                    SuppressedNode
                      Call Poner_broca
          Popup Message (haltProgram=false message=Linea17 con chica Terminada! inputType=Text)
          Folder Linea18
            Folder Marcar_puntos
              MoveL speed 100 mm/s, acceleration 500 mm/s^2 (useActiveTCP=true) feature=Base
                Waypoint Linea18_A: TCP in base x=-658.633 y=625.71 z=110.713 mm, rx=-0.2145 ry=-3.1278 rz=-0.004 rad; joints [-48.425, -62.133, 90.617, -28.11, -229.743, 0.749] deg; TCP offset x=0.411 y=-218.298 z=37.994 mm, rx=1.558 ry=-0.1255 rz=0.1212 rad
                Waypoint Linea18_B: TCP in base x=-1149.609 y=625.735 z=110.055 mm, rx=1.1641 ry=-2.9058 rz=0.0105 rad; joints [-36.269, -18.655, 11.335, 7.818, -269.001, 0.894] deg
            Folder AB
              'desbaste_inicial'
              bajada_broca := p[0,0,-0.008,0,0,0]
              barrenos_menos1 := 19
              barreno_actual := 0
              Loop While (checkContinuously=false) expression=barreno_actual≤barrenos_menos1
                Folder Perforacion
                  MoveL speed 100 mm/s, acceleration 500 mm/s^2 (useActiveTCP=true) feature=Base
                    If barreno_actual≟6  or barreno_actual≟13
                      barreno_actual := barreno_actual+1
                    internos := interpolate_pose(Linea18_A, Linea18_B, barreno_actual/barrenos_menos1)
                    Waypoint Waypoint (Variable): variable=internos
                    'desbaste_inicial'
                    bajada_broca := p[0,0,-0.008,0,0,0]
                    bajada := p[0,0,0.008,0,0,0]
                    MoveDirectionNode (selectedDirection=ZMinus toolParams=0.1, 0.15)
                      Until DISTANCE (allowActions=false deceleration=3 distanceNodeType=STOP) Distance=0.071; motionParameters(blendRadius=0)
                    MoveDirectionNode (selectedDirection=ZMinus toolParams=0.001, 0.001)
                      Until TOOL_CONTACT_DETECTION (allowActions=false retraction=0 decelerationAcceleration=0.001 decelerationAngularAcceleration=34.906585)
                    Popup Message (haltProgram=false message=punto contacto alanzdo inputType=Text)
                    MoveDirectionNode (selectedDirection=ZPlus toolParams=0.003, 0.005)
                      Until DISTANCE (allowActions=false deceleration=3 distanceNodeType=STOP) Distance=0.002; motionParameters(blendRadius=0)
                    Wait Sleep waitTime=0.3
                    Set DigitalOutput pin=config_out[1]; digitalValue=1
                    Wait Sleep waitTime=0.3
                    SuppressedNode
                      Loop Counting (count=3) loopVariable=Loop_92
                        bajar := pose_add(get_actual_tcp_pose(), bajada_broca)
                        Waypoint Waypoint (Variable): motionParameters(jointSpeed=1.047198 jointAcceleration=1.396263 cartesianSpeed=0.001 cartesianAcceleration=0.005); variable=bajar
                        subir := pose_sub(get_actual_tcp_pose(), bajada_broca)
                        Waypoint Waypoint (Variable): motionParameters(jointSpeed=1.047198 jointAcceleration=1.396263 cartesianSpeed=0.005 cartesianAcceleration=0.01); variable=subir
                        bajada_broca := pose_sub(bajada_broca, bajada)
                    MoveDirectionNode (selectedDirection=ZPlus toolParams=0.1, 0.15)
                      Until DISTANCE (allowActions=false deceleration=3 distanceNodeType=STOP) Distance=0.08; motionParameters(blendRadius=0)
                    Set DigitalOutput pin=config_out[1]; digitalValue=0
                    barreno_actual := barreno_actual+1
                    SuppressedNode
                      Call Quitar_broca
                    SuppressedNode
                      Call Poner_broca
          Popup Message (haltProgram=false message=Linea18 con chica Terminada! inputType=Text)
      Folder Broca_1
        Folder Linea7
          Folder Marcar_puntos
            MoveL speed 100 mm/s, acceleration 500 mm/s^2 (useActiveTCP=true) feature=Base
              Waypoint Home2: TCP in base x=-476.229 y=0 z=568.737 mm, rx=2.0263 ry=-2.3929 rz=-0.0208 rad; joints [-32.551, -116.469, 98.413, 17.843, -302.102, -0.163] deg; TCP offset x=0.411 y=-218.298 z=37.994 mm, rx=1.558 ry=-0.1255 rz=0.1212 rad
              Waypoint Linea7_A: TCP in base x=-749.561 y=-351.839 z=110.843 mm, rx=3.1084 ry=-0.3759 rz=-0.0174 rad; joints [1.917, -65.95, 96.598, -30.808, -353.455, -0.309] deg
              Folder bajada_comprobacion
                MoveDirectionNode (selectedDirection=ZMinus toolParams=0.1, 0.15)
                  Until DISTANCE (allowActions=false deceleration=3 distanceNodeType=STOP) Distance=0.071; motionParameters(blendRadius=0)
                MoveDirectionNode (selectedDirection=ZMinus toolParams=0.007, 0.007)
                  Until TOOL_CONTACT_DETECTION (allowActions=false retraction=0 decelerationAcceleration=0.02 decelerationAngularAcceleration=34.906585)
                MoveDirectionNode (selectedDirection=ZPlus toolParams=0.1, 0.15)
                  Until DISTANCE (allowActions=false deceleration=3 distanceNodeType=STOP) Distance=0.08; motionParameters(blendRadius=0)
              Waypoint Linea7_B: TCP in base x=-795.37 y=-351.638 z=110.748 mm, rx=3.1084 ry=-0.3758 rz=-0.0174 rad; joints [1.792, -62.243, 90.906, -28.822, -353.578, -0.309] deg
              Folder bajada_comprobacion
                MoveDirectionNode (selectedDirection=ZMinus toolParams=0.1, 0.15)
                  Until DISTANCE (allowActions=false deceleration=3 distanceNodeType=STOP) Distance=0.071; motionParameters(blendRadius=0)
                MoveDirectionNode (selectedDirection=ZMinus toolParams=0.007, 0.007)
                  Until TOOL_CONTACT_DETECTION (allowActions=false retraction=0 decelerationAcceleration=0.02 decelerationAngularAcceleration=34.906585)
                MoveDirectionNode (selectedDirection=ZPlus toolParams=0.1, 0.15)
                  Until DISTANCE (allowActions=false deceleration=3 distanceNodeType=STOP) Distance=0.08; motionParameters(blendRadius=0)
          Folder AB
            'desbaste_inicial'
            bajada_broca := p[0,0,-0.008,0,0,0]
            barrenos_menos1 := 2
            barreno_actual := 0
            Loop While (checkContinuously=false) expression=barreno_actual≤barrenos_menos1
              Folder Perforacion
                MoveL speed 100 mm/s, acceleration 500 mm/s^2 (useActiveTCP=true) feature=Base
                  internos := interpolate_pose(Linea7_A, Linea7_B, barreno_actual/barrenos_menos1)
                  Waypoint Waypoint (Variable): variable=internos
                  'desbaste_inicial'
                  bajada_broca := p[0,0,-0.024,0,0,0]
                  bajada := p[0,0,0.024,0,0,0]
                  MoveDirectionNode (selectedDirection=ZMinus toolParams=0.1, 0.15)
                    Until DISTANCE (allowActions=false deceleration=3 distanceNodeType=STOP) Distance=0.071; motionParameters(blendRadius=0)
                  MoveDirectionNode (selectedDirection=ZMinus toolParams=0.007, 0.007)
                    Until TOOL_CONTACT_DETECTION (allowActions=false retraction=0 decelerationAcceleration=0.02 decelerationAngularAcceleration=34.906585)
                  Popup Message (haltProgram=false message=punto contacto alanzdo inputType=Text)
                  MoveDirectionNode (selectedDirection=ZPlus toolParams=0.003, 0.005)
                    Until DISTANCE (allowActions=false deceleration=3 distanceNodeType=STOP) Distance=0.002; motionParameters(blendRadius=0)
                  Wait Sleep waitTime=0.3
                  Set DigitalOutput pin=config_out[1]; digitalValue=1
                  Wait Sleep waitTime=0.3
                  Loop Counting (count=1) loopVariable(name=Loop_96)
                    bajar := pose_add(get_actual_tcp_pose(), bajada_broca)
                    Waypoint Waypoint (Variable): motionParameters(jointSpeed=1.047198 jointAcceleration=1.396263 cartesianSpeed=0.01 cartesianAcceleration=0.01); variable=bajar
                    subir := pose_sub(get_actual_tcp_pose(), bajada_broca)
                    Waypoint Waypoint (Variable): motionParameters(jointSpeed=1.047198 jointAcceleration=1.396263 cartesianSpeed=0.015 cartesianAcceleration=0.015); variable=subir
                    bajada_broca := pose_sub(bajada_broca, bajada)
                  MoveDirectionNode (selectedDirection=ZPlus toolParams=0.1, 0.15)
                    Until DISTANCE (allowActions=false deceleration=3 distanceNodeType=STOP) Distance=0.08; motionParameters(blendRadius=0)
                  Set DigitalOutput pin=config_out[1]; digitalValue=0
                  barreno_actual := barreno_actual+1
                  Call Quitar_broca
                  Call Poner_broca
        Popup Message (haltProgram=false message=Linea7 con chica Terminada! inputType=Text)
        Folder Linea8
          Folder Marcar_puntos
            MoveL speed 100 mm/s, acceleration 500 mm/s^2 (useActiveTCP=true) feature=Base
              Waypoint Linea8_A: TCP in base x=-897.665 y=-351.421 z=110.406 mm, rx=3.1084 ry=-0.3758 rz=-0.0174 rad; joints [1.574, -53.621, 76.868, -23.4, -353.783, -0.317] deg; TCP offset x=0.411 y=-218.298 z=37.994 mm, rx=1.558 ry=-0.1255 rz=0.1212 rad
              Folder bajada_comprobacion
                MoveDirectionNode (selectedDirection=ZMinus toolParams=0.1, 0.15)
                  Until DISTANCE (allowActions=false deceleration=3 distanceNodeType=STOP) Distance=0.071; motionParameters(blendRadius=0)
                MoveDirectionNode (selectedDirection=ZMinus toolParams=0.007, 0.007)
                  Until TOOL_CONTACT_DETECTION (allowActions=false retraction=0 decelerationAcceleration=0.007 decelerationAngularAcceleration=34.906585)
                MoveDirectionNode (selectedDirection=ZPlus toolParams=0.1, 0.15)
                  Until DISTANCE (allowActions=false deceleration=3 distanceNodeType=STOP) Distance=0.08; motionParameters(blendRadius=0)
              Waypoint Linea8_B: TCP in base x=-1021.743 y=-350.913 z=110.77 mm, rx=3.1084 ry=-0.3758 rz=-0.0173 rad; joints [1.351, -41.656, 55.75, -14.225, -353.984, -0.335] deg; TCP offset x=0.411 y=-218.298 z=37.994 mm, rx=1.558 ry=-0.1255 rz=0.1212 rad
              Folder bajada_comprobacion
                MoveDirectionNode (selectedDirection=ZMinus toolParams=0.1, 0.15)
                  Until DISTANCE (allowActions=false deceleration=3 distanceNodeType=STOP) Distance=0.071; motionParameters(blendRadius=0)
                MoveDirectionNode (selectedDirection=ZMinus toolParams=0.007, 0.007)
                  Until TOOL_CONTACT_DETECTION (allowActions=false retraction=0 decelerationAcceleration=0.007 decelerationAngularAcceleration=34.906585)
                MoveDirectionNode (selectedDirection=ZPlus toolParams=0.1, 0.15)
                  Until DISTANCE (allowActions=false deceleration=3 distanceNodeType=STOP) Distance=0.08; motionParameters(blendRadius=0)
          Folder AB
            'desbaste_inicial'
            bajada_broca := p[0,0,-0.008,0,0,0]
            barrenos_menos1 := 5
            barreno_actual := 0
            Loop While (checkContinuously=false) expression=barreno_actual≤barrenos_menos1
              Folder Perforacion
                MoveL speed 100 mm/s, acceleration 500 mm/s^2 (useActiveTCP=true) feature=Base
                  internos := interpolate_pose(Linea8_A, Linea8_B, barreno_actual/barrenos_menos1)
                  Waypoint Waypoint (Variable): variable=internos
                  'desbaste_inicial'
                  bajada_broca := p[0,0,-0.024,0,0,0]
                  bajada := p[0,0,0.0024,0,0,0]
                  MoveDirectionNode (selectedDirection=ZMinus toolParams=0.1, 0.15)
                    Until DISTANCE (allowActions=false deceleration=3 distanceNodeType=STOP) Distance=0.071; motionParameters(blendRadius=0)
                  MoveDirectionNode (selectedDirection=ZMinus toolParams=0.01, 0.01)
                    Until TOOL_CONTACT_DETECTION (allowActions=false retraction=0 decelerationAcceleration=0.01 decelerationAngularAcceleration=34.906585)
                  Popup Message (haltProgram=false message=punto contacto alanzdo inputType=Text)
                  MoveDirectionNode (selectedDirection=ZPlus toolParams=0.003, 0.005)
                    Until DISTANCE (allowActions=false deceleration=3 distanceNodeType=STOP) Distance=0.002; motionParameters(blendRadius=0)
                  Wait Sleep waitTime=0.3
                  Set DigitalOutput pin=config_out[1]; digitalValue=1
                  Wait Sleep waitTime=0.3
                  Loop Counting (count=1) loopVariable(name=Loop_110)
                    bajar := pose_add(get_actual_tcp_pose(), bajada_broca)
                    Waypoint Waypoint (Variable): motionParameters(jointSpeed=1.047198 jointAcceleration=1.396263 cartesianSpeed=0.01 cartesianAcceleration=0.01); variable=bajar
                    subir := pose_sub(get_actual_tcp_pose(), bajada_broca)
                    Waypoint Waypoint (Variable): motionParameters(jointSpeed=1.047198 jointAcceleration=1.396263 cartesianSpeed=0.015 cartesianAcceleration=0.015); variable=subir
                    bajada_broca := pose_sub(bajada_broca, bajada)
                  MoveDirectionNode (selectedDirection=ZPlus toolParams=0.1, 0.15)
                    Until DISTANCE (allowActions=false deceleration=3 distanceNodeType=STOP) Distance=0.08; motionParameters(blendRadius=0)
                  Set DigitalOutput pin=config_out[1]; digitalValue=0
                  barreno_actual := barreno_actual+1
                  Call Quitar_broca
                  Call Poner_broca
        Popup Message (haltProgram=false message=Linea8 con chica Terminada! inputType=Text)
        Folder Linea9
          Folder Marcar_puntos
            MoveL speed 100 mm/s, acceleration 500 mm/s^2 (useActiveTCP=true) feature=Base
              Waypoint Linea9_A: TCP in base x=-1101.64 y=-350.63 z=110.828 mm, rx=3.1084 ry=-0.3759 rz=-0.0174 rad; joints [1.234, -31.471, 36.669, -5.317, -354.073, -0.351] deg; TCP offset x=0.411 y=-218.298 z=37.994 mm, rx=1.558 ry=-0.1255 rz=0.1212 rad
              Folder bajada_comprobacion
                MoveDirectionNode (selectedDirection=ZMinus toolParams=0.1, 0.15)
                  Until DISTANCE (allowActions=false deceleration=3 distanceNodeType=STOP) Distance=0.071; motionParameters(blendRadius=0)
                MoveDirectionNode (selectedDirection=ZMinus toolParams=0.007, 0.007)
                  Until TOOL_CONTACT_DETECTION (allowActions=false retraction=0 decelerationAcceleration=0.007 decelerationAngularAcceleration=34.906585)
                MoveDirectionNode (selectedDirection=ZPlus toolParams=0.1, 0.15)
                  Until DISTANCE (allowActions=false deceleration=3 distanceNodeType=STOP) Distance=0.08; motionParameters(blendRadius=0)
              Waypoint Linea9_B: TCP in base x=-1151.202 y=-350.816 z=110.405 mm, rx=3.1084 ry=-0.3759 rz=-0.0174 rad; joints [1.184, -21.077, 16.327, 4.623, -354.093, -0.341] deg
              Folder bajada_comprobacion
                MoveDirectionNode (selectedDirection=ZMinus toolParams=0.1, 0.15)
                  Until DISTANCE (allowActions=false deceleration=3 distanceNodeType=STOP) Distance=0.071; motionParameters(blendRadius=0)
                MoveDirectionNode (selectedDirection=ZMinus toolParams=0.007, 0.007)
                  Until TOOL_CONTACT_DETECTION (allowActions=false retraction=0 decelerationAcceleration=0.007 decelerationAngularAcceleration=34.906585)
                MoveDirectionNode (selectedDirection=ZPlus toolParams=0.1, 0.15)
                  Until DISTANCE (allowActions=false deceleration=3 distanceNodeType=STOP) Distance=0.08; motionParameters(blendRadius=0)
          Folder AB
            'desbaste_inicial'
            bajada_broca := p[0,0,-0.008,0,0,0]
            barrenos_menos1 := 2
            barreno_actual := 2
            Loop While (checkContinuously=false) expression=barreno_actual≤barrenos_menos1
              Folder Perforacion
                MoveL speed 100 mm/s, acceleration 500 mm/s^2 (useActiveTCP=true) feature=Base
                  internos := interpolate_pose(Linea9_A, Linea9_B, barreno_actual/barrenos_menos1)
                  Waypoint Waypoint (Variable): variable=internos
                  'desbaste_inicial'
                  bajada_broca := p[0,0,-0.024,0,0,0]
                  bajada := p[0,0,0.024,0,0,0]
                  MoveDirectionNode (selectedDirection=ZMinus toolParams=0.1, 0.15)
                    Until DISTANCE (allowActions=false deceleration=3 distanceNodeType=STOP) Distance=0.071; motionParameters(blendRadius=0)
                  MoveDirectionNode (selectedDirection=ZMinus toolParams=0.01, 0.01)
                    Until TOOL_CONTACT_DETECTION (allowActions=false retraction=0 decelerationAcceleration=0.01 decelerationAngularAcceleration=34.906585)
                  Popup Message (haltProgram=false message=punto contacto alanzdo inputType=Text)
                  MoveDirectionNode (selectedDirection=ZPlus toolParams=0.015, 0.015)
                    Until DISTANCE (allowActions=false deceleration=3 distanceNodeType=STOP) Distance=0.007; motionParameters(blendRadius=0)
                  Wait Sleep waitTime=0.3
                  Set DigitalOutput pin=config_out[1]; digitalValue=1
                  Wait Sleep waitTime=0.3
                  Loop Counting (count=1) loopVariable(name=Loop_114)
                    bajar := pose_add(get_actual_tcp_pose(), bajada_broca)
                    Waypoint Waypoint (Variable): motionParameters(jointSpeed=1.047198 jointAcceleration=1.396263 cartesianSpeed=0.01 cartesianAcceleration=0.01); variable=bajar
                    subir := pose_sub(get_actual_tcp_pose(), bajada_broca)
                    MoveDirectionNode (selectedDirection=ZPlus)
                      Until DISTANCE (allowActions=false deceleration=3 distanceNodeType=STOP) Distance=0.002; motionParameters(blendRadius=0)
                    Set DigitalOutput pin=config_out[1]; digitalValue=0
                    Waypoint Waypoint (Variable): motionParameters(jointSpeed=1.047198 jointAcceleration=1.396263 cartesianSpeed=0.015 cartesianAcceleration=0.015); variable=subir
                    bajada_broca := pose_sub(bajada_broca, bajada)
                  MoveDirectionNode (selectedDirection=ZPlus toolParams=0.1, 0.15)
                    Until DISTANCE (allowActions=false deceleration=3 distanceNodeType=STOP) Distance=0.08; motionParameters(blendRadius=0)
                  Set DigitalOutput pin=config_out[1]; digitalValue=0
                  barreno_actual := barreno_actual+1
                  Call Quitar_broca
                  Call Poner_broca
        Popup Message (haltProgram=false message=Linea9 con chica Terminada! inputType=Text)
        Folder Linea10
          Folder Marcar_puntos
            MoveL speed 100 mm/s, acceleration 500 mm/s^2 (useActiveTCP=true) feature=Base
              Waypoint Home2: TCP in base x=-476.229 y=0 z=568.737 mm, rx=2.0263 ry=-2.3929 rz=-0.0208 rad; joints [-32.551, -116.469, 98.413, 17.843, -302.102, -0.163] deg; TCP offset x=0.411 y=-218.298 z=37.994 mm, rx=1.558 ry=-0.1255 rz=0.1212 rad
              Waypoint Linea10_A: TCP in base x=-633.308 y=-317.691 z=110.995 mm, rx=3.1084 ry=-0.3759 rz=-0.0173 rad; joints [-0.882, -76.128, 110.969, -35.097, -356.258, -0.208] deg
              Folder bajada_comprobacion
                MoveDirectionNode (selectedDirection=ZMinus toolParams=0.1, 0.15)
                  Until DISTANCE (allowActions=false deceleration=3 distanceNodeType=STOP) Distance=0.071; motionParameters(blendRadius=0)
                MoveDirectionNode (selectedDirection=ZMinus toolParams=0.007, 0.007)
                  Until TOOL_CONTACT_DETECTION (allowActions=false retraction=0 decelerationAcceleration=0.02 decelerationAngularAcceleration=34.906585)
                MoveDirectionNode (selectedDirection=ZPlus toolParams=0.1, 0.15)
                  Until DISTANCE (allowActions=false deceleration=3 distanceNodeType=STOP) Distance=0.08; motionParameters(blendRadius=0)
              Waypoint Linea10_B: TCP in base x=-636.724 y=-266.696 z=110.314 mm, rx=2.0205 ry=-2.3939 rz=-0.0206 rad; joints [10.675, -83.921, 120.731, -37.208, -258.826, -0.176] deg
              Folder bajada_comprobacion
                MoveDirectionNode (selectedDirection=ZMinus toolParams=0.1, 0.15)
                  Until DISTANCE (allowActions=false deceleration=3 distanceNodeType=STOP) Distance=0.071; motionParameters(blendRadius=0)
                MoveDirectionNode (selectedDirection=ZMinus toolParams=0.007, 0.007)
                  Until TOOL_CONTACT_DETECTION (allowActions=false retraction=0 decelerationAcceleration=0.02 decelerationAngularAcceleration=34.906585)
                MoveDirectionNode (selectedDirection=ZPlus toolParams=0.1, 0.15)
                  Until DISTANCE (allowActions=false deceleration=3 distanceNodeType=STOP) Distance=0.08; motionParameters(blendRadius=0)
          Folder AB
            'desbaste_inicial'
            bajada_broca := p[0,0,-0.008,0,0,0]
            barrenos_menos1 := 2
            barreno_actual := 0
            Loop While (checkContinuously=false) expression=barreno_actual≤barrenos_menos1
              Folder Perforacion
                MoveL speed 100 mm/s, acceleration 500 mm/s^2 (useActiveTCP=true) feature=Base
                  internos := interpolate_pose(Linea10_A, Linea10_B, barreno_actual/barrenos_menos1)
                  Waypoint Waypoint (Variable): variable=internos
                  'desbaste_inicial'
                  bajada_broca := p[0,0,-0.024,0,0,0]
                  bajada := p[0,0,0.024,0,0,0]
                  MoveDirectionNode (selectedDirection=ZMinus toolParams=0.1, 0.15)
                    Until DISTANCE (allowActions=false deceleration=3 distanceNodeType=STOP) Distance=0.071; motionParameters(blendRadius=0)
                  MoveDirectionNode (selectedDirection=ZMinus toolParams=0.007, 0.007)
                    Until TOOL_CONTACT_DETECTION (allowActions=false retraction=0 decelerationAcceleration=0.02 decelerationAngularAcceleration=34.906585)
                  Popup Message (haltProgram=false message=punto contacto alanzdo inputType=Text)
                  MoveDirectionNode (selectedDirection=ZPlus toolParams=0.015, 0.015)
                    Until DISTANCE (allowActions=false deceleration=3 distanceNodeType=STOP) Distance=0.007; motionParameters(blendRadius=0)
                  Wait Sleep waitTime=0.3
                  Set DigitalOutput pin=config_out[1]; digitalValue=1
                  Wait Sleep waitTime=0.3
                  Loop Counting (count=1) loopVariable(name=Loop_118)
                    bajar := pose_add(get_actual_tcp_pose(), bajada_broca)
                    Waypoint Waypoint (Variable): motionParameters(jointSpeed=1.047198 jointAcceleration=1.396263 cartesianSpeed=0.004 cartesianAcceleration=0.004); variable=bajar
                    subir := pose_sub(get_actual_tcp_pose(), bajada_broca)
                    MoveDirectionNode (selectedDirection=ZPlus toolParams=0.015, 0.015)
                      Until DISTANCE (allowActions=false deceleration=3 distanceNodeType=STOP) Distance=0.002; motionParameters(blendRadius=0)
                    Set DigitalOutput pin=config_out[1]; digitalValue=0
                    Waypoint Waypoint (Variable): motionParameters(jointSpeed=1.047198 jointAcceleration=1.396263 cartesianSpeed=0.015 cartesianAcceleration=0.015); variable=subir
                    bajada_broca := pose_sub(bajada_broca, bajada)
                  MoveDirectionNode (selectedDirection=ZPlus toolParams=0.1, 0.15)
                    Until DISTANCE (allowActions=false deceleration=3 distanceNodeType=STOP) Distance=0.08; motionParameters(blendRadius=0)
                  Set DigitalOutput pin=config_out[1]; digitalValue=0
                  barreno_actual := barreno_actual+1
                  SuppressedNode
                    Call Quitar_broca
                  SuppressedNode
                    Call Poner_broca
        Popup Message (haltProgram=false message=Linea10 con chica Terminada! inputType=Text)
        Folder Linea11
          Folder Marcar_puntos
            MoveL speed 100 mm/s, acceleration 500 mm/s^2 (useActiveTCP=true) feature=Base
              Waypoint Linea11_A: TCP in base x=-635.968 y=-137.768 z=110.292 mm, rx=2.0222 ry=-2.396 rz=-0.017 rad; joints [-4.214, -88.643, 125.799, -37.329, -273.711, -0.094] deg; TCP offset x=0.411 y=-218.298 z=37.994 mm, rx=1.558 ry=-0.1255 rz=0.1212 rad
              Folder bajada_comprobacion
                MoveDirectionNode (selectedDirection=ZMinus toolParams=0.1, 0.15)
                  Until DISTANCE (allowActions=false deceleration=3 distanceNodeType=STOP) Distance=0.071; motionParameters(blendRadius=0)
                MoveDirectionNode (selectedDirection=ZMinus toolParams=0.007, 0.007)
                  Until TOOL_CONTACT_DETECTION (allowActions=false retraction=0 decelerationAcceleration=0.02 decelerationAngularAcceleration=34.906585)
                MoveDirectionNode (selectedDirection=ZPlus toolParams=0.1, 0.15)
                  Until DISTANCE (allowActions=false deceleration=3 distanceNodeType=STOP) Distance=0.08; motionParameters(blendRadius=0)
              Waypoint Linea11_B: TCP in base x=-635.824 y=-83.112 z=110.948 mm, rx=2.0204 ry=-2.3939 rz=-0.0206 rad; joints [-10.934, -90.004, 127.169, -37.541, -280.432, -0.033] deg
              Folder bajada_comprobacion
                MoveDirectionNode (selectedDirection=ZMinus toolParams=0.1, 0.15)
                  Until DISTANCE (allowActions=false deceleration=3 distanceNodeType=STOP) Distance=0.071; motionParameters(blendRadius=0)
                MoveDirectionNode (selectedDirection=ZMinus toolParams=0.007, 0.007)
                  Until TOOL_CONTACT_DETECTION (allowActions=false retraction=0 decelerationAcceleration=0.02 decelerationAngularAcceleration=34.906585)
                MoveDirectionNode (selectedDirection=ZPlus toolParams=0.1, 0.15)
                  Until DISTANCE (allowActions=false deceleration=3 distanceNodeType=STOP) Distance=0.08; motionParameters(blendRadius=0)
          Folder AB
            'desbaste_inicial'
            bajada_broca := p[0,0,-0.008,0,0,0]
            barrenos_menos1 := 2
            barreno_actual := 0
            Loop While (checkContinuously=false) expression=barreno_actual≤barrenos_menos1
              Folder Perforacion
                MoveL speed 100 mm/s, acceleration 500 mm/s^2 (useActiveTCP=true) feature=Base
                  SuppressedNode
                    If barreno_actual≟5
                      barreno_actual := barreno_actual+1
                  internos := interpolate_pose(Linea11_A, Linea11_B, barreno_actual/barrenos_menos1)
                  Waypoint Waypoint (Variable): variable=internos
                  'desbaste_inicial'
                  bajada_broca := p[0,0,-0.024,0,0,0]
                  bajada := p[0,0,0.024,0,0,0]
                  MoveDirectionNode (selectedDirection=ZMinus toolParams=0.1, 0.15)
                    Until DISTANCE (allowActions=false deceleration=3 distanceNodeType=STOP) Distance=0.071; motionParameters(blendRadius=0)
                  MoveDirectionNode (selectedDirection=ZMinus toolParams=0.007, 0.007)
                    Until TOOL_CONTACT_DETECTION (allowActions=false retraction=0 decelerationAcceleration=0.02 decelerationAngularAcceleration=34.906585)
                  Popup Message (haltProgram=false message=punto contacto alanzdo inputType=Text)
                  MoveDirectionNode (selectedDirection=ZPlus toolParams=0.015, 0.015)
                    Until DISTANCE (allowActions=false deceleration=3 distanceNodeType=STOP) Distance=0.007; motionParameters(blendRadius=0)
                  Wait Sleep waitTime=0.3
                  Set DigitalOutput pin=config_out[1]; digitalValue=1
                  Wait Sleep waitTime=0.3
                  Loop Counting (count=1) loopVariable(name=Loop_122)
                    bajar := pose_add(get_actual_tcp_pose(), bajada_broca)
                    Waypoint Waypoint (Variable): motionParameters(jointSpeed=1.047198 jointAcceleration=1.396263 cartesianSpeed=0.004 cartesianAcceleration=0.004); variable=bajar
                    subir := pose_sub(get_actual_tcp_pose(), bajada_broca)
                    MoveDirectionNode (selectedDirection=ZPlus toolParams=0.015, 0.015)
                      Until DISTANCE (allowActions=false deceleration=3 distanceNodeType=STOP) Distance=0.002; motionParameters(blendRadius=0)
                    Set DigitalOutput pin=config_out[1]; digitalValue=0
                    Waypoint Waypoint (Variable): motionParameters(jointSpeed=1.047198 jointAcceleration=1.396263 cartesianSpeed=0.015 cartesianAcceleration=0.015); variable=subir
                    bajada_broca := pose_sub(bajada_broca, bajada)
                  MoveDirectionNode (selectedDirection=ZPlus toolParams=0.1, 0.15)
                    Until DISTANCE (allowActions=false deceleration=3 distanceNodeType=STOP) Distance=0.08; motionParameters(blendRadius=0)
                  Set DigitalOutput pin=config_out[1]; digitalValue=0
                  barreno_actual := barreno_actual+1
                  SuppressedNode
                    Call Quitar_broca
                  SuppressedNode
                    Call Poner_broca
        Popup Message (haltProgram=false message=Linea11 con chica Terminada! inputType=Text)
        Folder Linea12
          Folder Marcar_puntos
            MoveL speed 100 mm/s, acceleration 500 mm/s^2 (useActiveTCP=true) feature=Base
              Waypoint Linea12_A: TCP in base x=-635.349 y=-59.56 z=110.675 mm, rx=2.0204 ry=-2.3939 rz=-0.0205 rad; joints [-13.849, -90.386, 127.583, -37.571, -283.348, -0.016] deg
              Folder bajada_comprobacion
                MoveDirectionNode (selectedDirection=ZMinus toolParams=0.1, 0.15)
                  Until DISTANCE (allowActions=false deceleration=3 distanceNodeType=STOP) Distance=0.071; motionParameters(blendRadius=0)
                MoveDirectionNode (selectedDirection=ZMinus toolParams=0.007, 0.007)
                  Until TOOL_CONTACT_DETECTION (allowActions=false retraction=0 decelerationAcceleration=0.02 decelerationAngularAcceleration=34.906585)
                MoveDirectionNode (selectedDirection=ZPlus toolParams=0.1, 0.15)
                  Until DISTANCE (allowActions=false deceleration=3 distanceNodeType=STOP) Distance=0.08; motionParameters(blendRadius=0)
              Waypoint Linea12_B: TCP in base x=-634.713 y=114.181 z=110.553 mm, rx=2.0204 ry=-2.3939 rz=-0.0206 rad; joints [-33.919, -89.532, 126.745, -37.627, -303.419, 0.135] deg
              Folder bajada_comprobacion
                MoveDirectionNode (selectedDirection=ZMinus toolParams=0.1, 0.15)
                  Until DISTANCE (allowActions=false deceleration=3 distanceNodeType=STOP) Distance=0.071; motionParameters(blendRadius=0)
                MoveDirectionNode (selectedDirection=ZMinus toolParams=0.007, 0.007)
                  Until TOOL_CONTACT_DETECTION (allowActions=false retraction=0 decelerationAcceleration=0.02 decelerationAngularAcceleration=34.906585)
                MoveDirectionNode (selectedDirection=ZPlus toolParams=0.1, 0.15)
                  Until DISTANCE (allowActions=false deceleration=3 distanceNodeType=STOP) Distance=0.08; motionParameters(blendRadius=0)
          Folder AB
            'desbaste_inicial'
            bajada_broca := p[0,0,-0.008,0,0,0]
            barrenos_menos1 := 7
            barreno_actual := 0
            Loop While (checkContinuously=false) expression=barreno_actual≤barrenos_menos1
              Folder Perforacion
                MoveL speed 100 mm/s, acceleration 500 mm/s^2 (useActiveTCP=true) feature=Base
                  If barreno_actual≟2
                    barreno_actual := barreno_actual+1
                  internos := interpolate_pose(Linea12_A, Linea12_B, barreno_actual/barrenos_menos1)
                  Waypoint Waypoint (Variable): variable=internos
                  'desbaste_inicial'
                  bajada_broca := p[0,0,-0.024,0,0,0]
                  bajada := p[0,0,0.024,0,0,0]
                  MoveDirectionNode (selectedDirection=ZMinus toolParams=0.1, 0.15)
                    Until DISTANCE (allowActions=false deceleration=3 distanceNodeType=STOP) Distance=0.071; motionParameters(blendRadius=0)
                  MoveDirectionNode (selectedDirection=ZMinus toolParams=0.007, 0.007)
                    Until TOOL_CONTACT_DETECTION (allowActions=false retraction=0 decelerationAcceleration=0.02 decelerationAngularAcceleration=34.906585)
                  Popup Message (haltProgram=false message=punto contacto alanzdo inputType=Text)
                  MoveDirectionNode (selectedDirection=ZPlus toolParams=0.003, 0.005)
                    Until DISTANCE (allowActions=false deceleration=3 distanceNodeType=STOP) Distance=0.002; motionParameters(blendRadius=0)
                  Wait Sleep waitTime=0.3
                  Set DigitalOutput pin=config_out[1]; digitalValue=1
                  Wait Sleep waitTime=0.3
                  Loop Counting (count=1) loopVariable(name=Loop_126)
                    bajar := pose_add(get_actual_tcp_pose(), bajada_broca)
                    Waypoint Waypoint (Variable): motionParameters(jointSpeed=1.047198 jointAcceleration=1.396263 cartesianSpeed=0.004 cartesianAcceleration=0.004); variable=bajar
                    subir := pose_sub(get_actual_tcp_pose(), bajada_broca)
                    MoveDirectionNode (selectedDirection=ZPlus toolParams=0.015, 0.015)
                      Until DISTANCE (allowActions=false deceleration=3 distanceNodeType=STOP) Distance=0.002; motionParameters(blendRadius=0)
                    Set DigitalOutput pin=config_out[1]; digitalValue=0
                    Waypoint Waypoint (Variable): motionParameters(jointSpeed=1.047198 jointAcceleration=1.396263 cartesianSpeed=0.015 cartesianAcceleration=0.015); variable=subir
                    bajada_broca := pose_sub(bajada_broca, bajada)
                  MoveDirectionNode (selectedDirection=ZPlus toolParams=0.1, 0.15)
                    Until DISTANCE (allowActions=false deceleration=3 distanceNodeType=STOP) Distance=0.08; motionParameters(blendRadius=0)
                  Set DigitalOutput pin=config_out[1]; digitalValue=0
                  barreno_actual := barreno_actual+1
                  SuppressedNode
                    Call Quitar_broca
                  SuppressedNode
                    Call Poner_broca
        Popup Message (haltProgram=false message=Linea12 con chica Terminada! inputType=Text)
        Folder Linea13
          Folder Marcar_puntos
            MoveL speed 100 mm/s, acceleration 500 mm/s^2 (useActiveTCP=true) feature=Base
              Waypoint Linea13_A: TCP in base x=-634.623 y=269.838 z=110.202 mm, rx=2.0205 ry=-2.3939 rz=-0.0206 rad; joints [-47.693, -84.101, 120.951, -37.343, -317.193, 0.28] deg
              Folder bajada_comprobacion
                MoveDirectionNode (selectedDirection=ZMinus toolParams=0.1, 0.15)
                  Until DISTANCE (allowActions=false deceleration=3 distanceNodeType=STOP) Distance=0.071; motionParameters(blendRadius=0)
                MoveDirectionNode (selectedDirection=ZMinus toolParams=0.007, 0.007)
                  Until TOOL_CONTACT_DETECTION (allowActions=false retraction=0 decelerationAcceleration=0.02 decelerationAngularAcceleration=34.906585)
                MoveDirectionNode (selectedDirection=ZPlus toolParams=0.1, 0.15)
                  Until DISTANCE (allowActions=false deceleration=3 distanceNodeType=STOP) Distance=0.08; motionParameters(blendRadius=0)
              Waypoint Linea13_B: TCP in base x=-634.043 y=326.314 z=110.496 mm, rx=2.0205 ry=-2.3939 rz=-0.0206 rad; joints [-51.641, -81.48, 117.853, -36.903, -321.141, 0.338] deg
              Folder bajada_comprobacion
                MoveDirectionNode (selectedDirection=ZMinus toolParams=0.1, 0.15)
                  Until DISTANCE (allowActions=false deceleration=3 distanceNodeType=STOP) Distance=0.071; motionParameters(blendRadius=0)
                MoveDirectionNode (selectedDirection=ZMinus toolParams=0.007, 0.007)
                  Until TOOL_CONTACT_DETECTION (allowActions=false retraction=0 decelerationAcceleration=0.02 decelerationAngularAcceleration=34.906585)
                MoveDirectionNode (selectedDirection=ZPlus toolParams=0.1, 0.15)
                  Until DISTANCE (allowActions=false deceleration=3 distanceNodeType=STOP) Distance=0.08; motionParameters(blendRadius=0)
          Folder AB
            'desbaste_inicial'
            bajada_broca := p[0,0,-0.008,0,0,0]
            barrenos_menos1 := 2
            barreno_actual := 0
            Loop While (checkContinuously=false) expression=barreno_actual≤barrenos_menos1
              Folder Perforacion
                MoveL speed 100 mm/s, acceleration 500 mm/s^2 (useActiveTCP=true) feature=Base
                  SuppressedNode
                    If barreno_actual≟2
                      barreno_actual := barreno_actual+1
                  internos := interpolate_pose(Linea13_A, Linea13_B, barreno_actual/barrenos_menos1)
                  Waypoint Waypoint (Variable): variable=internos
                  'desbaste_inicial'
                  bajada_broca := p[0,0,-0.024,0,0,0]
                  bajada := p[0,0,0.024,0,0,0]
                  MoveDirectionNode (selectedDirection=ZMinus toolParams=0.1, 0.15)
                    Until DISTANCE (allowActions=false deceleration=3 distanceNodeType=STOP) Distance=0.071; motionParameters(blendRadius=0)
                  MoveDirectionNode (selectedDirection=ZMinus toolParams=0.007, 0.007)
                    Until TOOL_CONTACT_DETECTION (allowActions=false retraction=0 decelerationAcceleration=0.02 decelerationAngularAcceleration=34.906585)
                  Popup Message (haltProgram=false message=punto contacto alanzdo inputType=Text)
                  MoveDirectionNode (selectedDirection=ZPlus toolParams=0.003, 0.005)
                    Until DISTANCE (allowActions=false deceleration=3 distanceNodeType=STOP) Distance=0.002; motionParameters(blendRadius=0)
                  Wait Sleep waitTime=0.3
                  Set DigitalOutput pin=config_out[1]; digitalValue=1
                  Wait Sleep waitTime=0.3
                  Loop Counting (count=1) loopVariable(name=Loop_129)
                    bajar := pose_add(get_actual_tcp_pose(), bajada_broca)
                    Waypoint Waypoint (Variable): motionParameters(jointSpeed=1.047198 jointAcceleration=1.396263 cartesianSpeed=0.004 cartesianAcceleration=0.004); variable=bajar
                    subir := pose_sub(get_actual_tcp_pose(), bajada_broca)
                    MoveDirectionNode (selectedDirection=ZPlus toolParams=0.015, 0.015)
                      Until DISTANCE (allowActions=false deceleration=3 distanceNodeType=STOP) Distance=0.002; motionParameters(blendRadius=0)
                    Set DigitalOutput pin=config_out[1]; digitalValue=0
                    Waypoint Waypoint (Variable): motionParameters(jointSpeed=1.047198 jointAcceleration=1.396263 cartesianSpeed=0.015 cartesianAcceleration=0.015); variable=subir
                    bajada_broca := pose_sub(bajada_broca, bajada)
                  MoveDirectionNode (selectedDirection=ZPlus toolParams=0.1, 0.15)
                    Until DISTANCE (allowActions=false deceleration=3 distanceNodeType=STOP) Distance=0.08; motionParameters(blendRadius=0)
                  Set DigitalOutput pin=config_out[1]; digitalValue=0
                  barreno_actual := barreno_actual+1
                  SuppressedNode
                    Call Quitar_broca
                  SuppressedNode
                    Call Poner_broca
        Popup Message (haltProgram=false message=Linea13 con chica Terminada! inputType=Text)
        Folder Linea14
          Folder Marcar_puntos
            MoveL speed 100 mm/s, acceleration 500 mm/s^2 (useActiveTCP=true) feature=Base
              Waypoint Linea14_A: TCP in base x=-633.963 y=349.887 z=111.384 mm, rx=2.0205 ry=-2.3938 rz=-0.0205 rad; joints [-53.122, -80.339, 116.362, -36.569, -322.623, 0.363] deg
              Folder bajada_comprobacion
                MoveDirectionNode (selectedDirection=ZMinus toolParams=0.1, 0.15)
                  Until DISTANCE (allowActions=false deceleration=3 distanceNodeType=STOP) Distance=0.071; motionParameters(blendRadius=0)
                MoveDirectionNode (selectedDirection=ZMinus toolParams=0.007, 0.007)
                  Until TOOL_CONTACT_DETECTION (allowActions=false retraction=0 decelerationAcceleration=0.02 decelerationAngularAcceleration=34.906585)
                MoveDirectionNode (selectedDirection=ZPlus toolParams=0.1, 0.15)
                  Until DISTANCE (allowActions=false deceleration=3 distanceNodeType=STOP) Distance=0.08; motionParameters(blendRadius=0)
              Waypoint Linea14_B: TCP in base x=-633.711 y=491.848 z=110.684 mm, rx=2.0205 ry=-2.3939 rz=-0.0205 rad; joints [-60.395, -72.347, 105.992, -34.301, -329.892, 0.503] deg
              Folder bajada_comprobacion
                MoveDirectionNode (selectedDirection=ZMinus toolParams=0.1, 0.15)
                  Until DISTANCE (allowActions=false deceleration=3 distanceNodeType=STOP) Distance=0.071; motionParameters(blendRadius=0)
                MoveDirectionNode (selectedDirection=ZMinus toolParams=0.007, 0.007)
                  Until TOOL_CONTACT_DETECTION (allowActions=false retraction=0 decelerationAcceleration=0.02 decelerationAngularAcceleration=34.906585)
                MoveDirectionNode (selectedDirection=ZPlus toolParams=0.1, 0.15)
                  Until DISTANCE (allowActions=false deceleration=3 distanceNodeType=STOP) Distance=0.08; motionParameters(blendRadius=0)
          Folder AB
            'desbaste_inicial'
            bajada_broca := p[0,0,-0.008,0,0,0]
            barrenos_menos1 := 5
            barreno_actual := 0
            Loop While (checkContinuously=false) expression=barreno_actual≤barrenos_menos1
              Folder Perforacion
                MoveL speed 100 mm/s, acceleration 500 mm/s^2 (useActiveTCP=true) feature=Base
                  If barreno_actual≟3
                    barreno_actual := barreno_actual+1
                  internos := interpolate_pose(Linea14_A, Linea14_B, barreno_actual/barrenos_menos1)
                  Waypoint Waypoint (Variable): variable=internos
                  'desbaste_inicial'
                  bajada_broca := p[0,0,-0.024,0,0,0]
                  bajada := p[0,0,0.024,0,0,0]
                  MoveDirectionNode (selectedDirection=ZMinus toolParams=0.1, 0.15)
                    Until DISTANCE (allowActions=false deceleration=3 distanceNodeType=STOP) Distance=0.071; motionParameters(blendRadius=0)
                  MoveDirectionNode (selectedDirection=ZMinus toolParams=0.007, 0.007)
                    Until TOOL_CONTACT_DETECTION (allowActions=false retraction=0 decelerationAcceleration=0.02 decelerationAngularAcceleration=34.906585)
                  Popup Message (haltProgram=false message=punto contacto alanzdo inputType=Text)
                  MoveDirectionNode (selectedDirection=ZPlus toolParams=0.003, 0.005)
                    Until DISTANCE (allowActions=false deceleration=3 distanceNodeType=STOP) Distance=0.002; motionParameters(blendRadius=0)
                  Wait Sleep waitTime=0.3
                  Set DigitalOutput pin=config_out[1]; digitalValue=1
                  Wait Sleep waitTime=0.3
                  Loop Counting (count=1) loopVariable(name=Loop_131)
                    bajar := pose_add(get_actual_tcp_pose(), bajada_broca)
                    Waypoint Waypoint (Variable): motionParameters(jointSpeed=1.047198 jointAcceleration=1.396263 cartesianSpeed=0.004 cartesianAcceleration=0.004); variable=bajar
                    subir := pose_sub(get_actual_tcp_pose(), bajada_broca)
                    MoveDirectionNode (selectedDirection=ZPlus toolParams=0.015, 0.015)
                      Until DISTANCE (allowActions=false deceleration=3 distanceNodeType=STOP) Distance=0.002; motionParameters(blendRadius=0)
                    Set DigitalOutput pin=config_out[1]; digitalValue=0
                    Waypoint Waypoint (Variable): motionParameters(jointSpeed=1.047198 jointAcceleration=1.396263 cartesianSpeed=0.015 cartesianAcceleration=0.015); variable=subir
                    bajada_broca := pose_sub(bajada_broca, bajada)
                  MoveDirectionNode (selectedDirection=ZPlus toolParams=0.1, 0.15)
                    Until DISTANCE (allowActions=false deceleration=3 distanceNodeType=STOP) Distance=0.08; motionParameters(blendRadius=0)
                  Set DigitalOutput pin=config_out[1]; digitalValue=0
                  barreno_actual := barreno_actual+1
                  SuppressedNode
                    Call Quitar_broca
                  SuppressedNode
                    Call Poner_broca
        Popup Message (haltProgram=false message=Linea14 con chica Terminada! inputType=Text)
        Folder Linea15
          Folder Marcar_puntos
            MoveL speed 100 mm/s, acceleration 500 mm/s^2 (useActiveTCP=true) feature=Base
              Waypoint Linea15_A: TCP in base x=-633.318 y=515.44 z=110.158 mm, rx=2.0204 ry=-2.394 rz=-0.0205 rad; joints [-61.401, -70.918, 104.049, -33.805, -330.892, 0.526] deg
              Folder bajada_comprobacion
                MoveDirectionNode (selectedDirection=ZMinus toolParams=0.1, 0.15)
                  Until DISTANCE (allowActions=false deceleration=3 distanceNodeType=STOP) Distance=0.071; motionParameters(blendRadius=0)
                MoveDirectionNode (selectedDirection=ZMinus toolParams=0.007, 0.007)
                  Until TOOL_CONTACT_DETECTION (allowActions=false retraction=0 decelerationAcceleration=0.02 decelerationAngularAcceleration=34.906585)
                MoveDirectionNode (selectedDirection=ZPlus toolParams=0.1, 0.15)
                  Until DISTANCE (allowActions=false deceleration=3 distanceNodeType=STOP) Distance=0.08; motionParameters(blendRadius=0)
              Waypoint Linea15_B: TCP in base x=-632.971 y=593.971 z=110.611 mm, rx=2.0204 ry=-2.3939 rz=-0.0206 rad; joints [-64.313, -66.034, 96.849, -31.559, -333.804, 0.606] deg
              Folder bajada_comprobacion
                MoveDirectionNode (selectedDirection=ZMinus toolParams=0.1, 0.15)
                  Until DISTANCE (allowActions=false deceleration=3 distanceNodeType=STOP) Distance=0.071; motionParameters(blendRadius=0)
                MoveDirectionNode (selectedDirection=ZMinus toolParams=0.007, 0.007)
                  Until TOOL_CONTACT_DETECTION (allowActions=false retraction=0 decelerationAcceleration=0.02 decelerationAngularAcceleration=34.906585)
                MoveDirectionNode (selectedDirection=ZPlus toolParams=0.1, 0.15)
                  Until DISTANCE (allowActions=false deceleration=3 distanceNodeType=STOP) Distance=0.08; motionParameters(blendRadius=0)
          Folder AB
            'desbaste_inicial'
            bajada_broca := p[0,0,-0.008,0,0,0]
            barrenos_menos1 := 3
            barreno_actual := 0
            Loop While (checkContinuously=false) expression=barreno_actual≤barrenos_menos1
              Folder Perforacion
                MoveL speed 100 mm/s, acceleration 500 mm/s^2 (useActiveTCP=true) feature=Base
                  SuppressedNode
                    If barreno_actual≟3
                      barreno_actual := barreno_actual+1
                  internos := interpolate_pose(Linea15_A, Linea15_B, barreno_actual/barrenos_menos1)
                  Waypoint Waypoint (Variable): variable=internos
                  'desbaste_inicial'
                  bajada_broca := p[0,0,-0.024,0,0,0]
                  bajada := p[0,0,0.024,0,0,0]
                  MoveDirectionNode (selectedDirection=ZMinus toolParams=0.1, 0.15)
                    Until DISTANCE (allowActions=false deceleration=3 distanceNodeType=STOP) Distance=0.071; motionParameters(blendRadius=0)
                  MoveDirectionNode (selectedDirection=ZMinus toolParams=0.007, 0.007)
                    Until TOOL_CONTACT_DETECTION (allowActions=false retraction=0 decelerationAcceleration=0.02 decelerationAngularAcceleration=34.906585)
                  Popup Message (haltProgram=false message=punto contacto alanzdo inputType=Text)
                  MoveDirectionNode (selectedDirection=ZPlus toolParams=0.003, 0.005)
                    Until DISTANCE (allowActions=false deceleration=3 distanceNodeType=STOP) Distance=0.002; motionParameters(blendRadius=0)
                  Wait Sleep waitTime=0.3
                  Set DigitalOutput pin=config_out[1]; digitalValue=1
                  Wait Sleep waitTime=0.3
                  Loop Counting (count=1) loopVariable(name=Loop_133)
                    bajar := pose_add(get_actual_tcp_pose(), bajada_broca)
                    Waypoint Waypoint (Variable): motionParameters(jointSpeed=1.047198 jointAcceleration=1.396263 cartesianSpeed=0.004 cartesianAcceleration=0.004); variable=bajar
                    subir := pose_sub(get_actual_tcp_pose(), bajada_broca)
                    MoveDirectionNode (selectedDirection=ZPlus toolParams=0.015, 0.015)
                      Until DISTANCE (allowActions=false deceleration=3 distanceNodeType=STOP) Distance=0.002; motionParameters(blendRadius=0)
                    Set DigitalOutput pin=config_out[1]; digitalValue=0
                    Waypoint Waypoint (Variable): motionParameters(jointSpeed=1.047198 jointAcceleration=1.396263 cartesianSpeed=0.015 cartesianAcceleration=0.015); variable=subir
                    bajada_broca := pose_sub(bajada_broca, bajada)
                  MoveDirectionNode (selectedDirection=ZPlus toolParams=0.1, 0.15)
                    Until DISTANCE (allowActions=false deceleration=3 distanceNodeType=STOP) Distance=0.08; motionParameters(blendRadius=0)
                  Set DigitalOutput pin=config_out[1]; digitalValue=0
                  barreno_actual := barreno_actual+1
                  SuppressedNode
                    Call Quitar_broca
                  SuppressedNode
                    Call Poner_broca
        Popup Message (haltProgram=false message=Linea15 con chica Terminada! inputType=Text)
        Folder Linea16
          Folder Marcar_puntos
            MoveL speed 100 mm/s, acceleration 500 mm/s^2 (useActiveTCP=true) feature=Base
              Waypoint Linea16_A: TCP in base x=-469.659 y=618.24 z=110.223 mm, rx=-0.2145 ry=-3.1278 rz=-0.004 rad; joints [-60.494, -74.578, 108.875, -33.964, -241.822, 0.658] deg
              Folder bajada_comprobacion
                MoveDirectionNode (selectedDirection=ZMinus toolParams=0.1, 0.15)
                  Until DISTANCE (allowActions=false deceleration=3 distanceNodeType=STOP) Distance=0.071; motionParameters(blendRadius=0)
                MoveDirectionNode (selectedDirection=ZMinus toolParams=0.007, 0.007)
                  Until TOOL_CONTACT_DETECTION (allowActions=false retraction=0 decelerationAcceleration=0.02 decelerationAngularAcceleration=34.906585)
                MoveDirectionNode (selectedDirection=ZPlus toolParams=0.1, 0.15)
                  Until DISTANCE (allowActions=false deceleration=3 distanceNodeType=STOP) Distance=0.08; motionParameters(blendRadius=0)
              Waypoint Linea16_B: TCP in base x=-493.719 y=618.586 z=110.183 mm, rx=-0.2145 ry=-3.1278 rz=-0.004 rad; joints [-58.661, -73.102, 106.872, -33.43, -239.985, 0.672] deg
              Folder bajada_comprobacion
                MoveDirectionNode (selectedDirection=ZMinus toolParams=0.1, 0.15)
                  Until DISTANCE (allowActions=false deceleration=3 distanceNodeType=STOP) Distance=0.071; motionParameters(blendRadius=0)
                MoveDirectionNode (selectedDirection=ZMinus toolParams=0.007, 0.007)
                  Until TOOL_CONTACT_DETECTION (allowActions=false retraction=0 decelerationAcceleration=0.02 decelerationAngularAcceleration=34.906585)
                MoveDirectionNode (selectedDirection=ZPlus toolParams=0.1, 0.15)
                  Until DISTANCE (allowActions=false deceleration=3 distanceNodeType=STOP) Distance=0.08; motionParameters(blendRadius=0)
          Folder AB
            'desbaste_inicial'
            bajada_broca := p[0,0,-0.008,0,0,0]
            barrenos_menos1 := 1
            barreno_actual := 0
            Loop While (checkContinuously=false) expression=barreno_actual≤barrenos_menos1
              Folder Perforacion
                MoveL speed 100 mm/s, acceleration 500 mm/s^2 (useActiveTCP=true) feature=Base
                  SuppressedNode
                    If barreno_actual≟3
                      barreno_actual := barreno_actual+1
                  internos := interpolate_pose(Linea16_A, Linea16_B, barreno_actual/barrenos_menos1)
                  Waypoint Waypoint (Variable): variable=internos
                  'desbaste_inicial'
                  bajada_broca := p[0,0,-0.024,0,0,0]
                  bajada := p[0,0,0.024,0,0,0]
                  MoveDirectionNode (selectedDirection=ZMinus toolParams=0.1, 0.15)
                    Until DISTANCE (allowActions=false deceleration=3 distanceNodeType=STOP) Distance=0.071; motionParameters(blendRadius=0)
                  MoveDirectionNode (selectedDirection=ZMinus toolParams=0.007, 0.007)
                    Until TOOL_CONTACT_DETECTION (allowActions=false retraction=0 decelerationAcceleration=0.02 decelerationAngularAcceleration=34.906585)
                  Popup Message (haltProgram=false message=punto contacto alanzdo inputType=Text)
                  MoveDirectionNode (selectedDirection=ZPlus toolParams=0.003, 0.005)
                    Until DISTANCE (allowActions=false deceleration=3 distanceNodeType=STOP) Distance=0.002; motionParameters(blendRadius=0)
                  Wait Sleep waitTime=0.3
                  Set DigitalOutput pin=config_out[1]; digitalValue=1
                  Wait Sleep waitTime=0.3
                  Loop Counting (count=1) loopVariable(name=Loop_135)
                    bajar := pose_add(get_actual_tcp_pose(), bajada_broca)
                    Waypoint Waypoint (Variable): motionParameters(jointSpeed=1.047198 jointAcceleration=1.396263 cartesianSpeed=0.004 cartesianAcceleration=0.004); variable=bajar
                    subir := pose_sub(get_actual_tcp_pose(), bajada_broca)
                    MoveDirectionNode (selectedDirection=ZPlus toolParams=0.015, 0.015)
                      Until DISTANCE (allowActions=false deceleration=3 distanceNodeType=STOP) Distance=0.002; motionParameters(blendRadius=0)
                    Set DigitalOutput pin=config_out[1]; digitalValue=0
                    Waypoint Waypoint (Variable): motionParameters(jointSpeed=1.047198 jointAcceleration=1.396263 cartesianSpeed=0.015 cartesianAcceleration=0.015); variable=subir
                    bajada_broca := pose_sub(bajada_broca, bajada)
                  MoveDirectionNode (selectedDirection=ZPlus toolParams=0.1, 0.15)
                    Until DISTANCE (allowActions=false deceleration=3 distanceNodeType=STOP) Distance=0.08; motionParameters(blendRadius=0)
                  Set DigitalOutput pin=config_out[1]; digitalValue=0
                  barreno_actual := barreno_actual+1
                  SuppressedNode
                    Call Quitar_broca
                  SuppressedNode
                    Call Poner_broca
        Popup Message (haltProgram=false message=Linea16 con chica Terminada! inputType=Text)
        Folder Linea17
          Folder Marcar_puntos
            MoveL speed 100 mm/s, acceleration 500 mm/s^2 (useActiveTCP=true) feature=Base
              Waypoint Linea17_A: TCP in base x=-523.229 y=618.283 z=110.575 mm, rx=-0.2145 ry=-3.1278 rz=-0.0039 rad; joints [-56.495, -71.324, 104.348, -32.678, -237.82, 0.686] deg
              Folder bajada_comprobacion
                MoveDirectionNode (selectedDirection=ZMinus toolParams=0.1, 0.15)
                  Until DISTANCE (allowActions=false deceleration=3 distanceNodeType=STOP) Distance=0.071; motionParameters(blendRadius=0)
                MoveDirectionNode (selectedDirection=ZMinus toolParams=0.007, 0.007)
                  Until TOOL_CONTACT_DETECTION (allowActions=false retraction=0 decelerationAcceleration=0.02 decelerationAngularAcceleration=34.906585)
                MoveDirectionNode (selectedDirection=ZPlus toolParams=0.1, 0.15)
                  Until DISTANCE (allowActions=false deceleration=3 distanceNodeType=STOP) Distance=0.08; motionParameters(blendRadius=0)
              Waypoint Linea17_B: TCP in base x=-574.505 y=618.78 z=110.128 mm, rx=-0.2145 ry=-3.1278 rz=-0.0039 rad; joints [-53.062, -68.029, 99.656, -31.269, -234.384, 0.712] deg
              Folder bajada_comprobacion
                MoveDirectionNode (selectedDirection=ZMinus toolParams=0.1, 0.15)
                  Until DISTANCE (allowActions=false deceleration=3 distanceNodeType=STOP) Distance=0.071; motionParameters(blendRadius=0)
                MoveDirectionNode (selectedDirection=ZMinus toolParams=0.007, 0.007)
                  Until TOOL_CONTACT_DETECTION (allowActions=false retraction=0 decelerationAcceleration=0.02 decelerationAngularAcceleration=34.906585)
                MoveDirectionNode (selectedDirection=ZPlus toolParams=0.1, 0.15)
                  Until DISTANCE (allowActions=false deceleration=3 distanceNodeType=STOP) Distance=0.08; motionParameters(blendRadius=0)
          Folder AB
            'desbaste_inicial'
            bajada_broca := p[0,0,-0.008,0,0,0]
            barrenos_menos1 := 2
            barreno_actual := 0
            Loop While (checkContinuously=false) expression=barreno_actual≤barrenos_menos1
              Folder Perforacion
                MoveL speed 100 mm/s, acceleration 500 mm/s^2 (useActiveTCP=true) feature=Base
                  SuppressedNode
                    If barreno_actual≟3
                      barreno_actual := barreno_actual+1
                  internos := interpolate_pose(Linea17_A, Linea17_B, barreno_actual/barrenos_menos1)
                  Waypoint Waypoint (Variable): variable=internos
                  'desbaste_inicial'
                  bajada_broca := p[0,0,-0.024,0,0,0]
                  bajada := p[0,0,0.024,0,0,0]
                  MoveDirectionNode (selectedDirection=ZMinus toolParams=0.1, 0.15)
                    Until DISTANCE (allowActions=false deceleration=3 distanceNodeType=STOP) Distance=0.071; motionParameters(blendRadius=0)
                  MoveDirectionNode (selectedDirection=ZMinus toolParams=0.007, 0.007)
                    Until TOOL_CONTACT_DETECTION (allowActions=false retraction=0 decelerationAcceleration=0.02 decelerationAngularAcceleration=34.906585)
                  Popup Message (haltProgram=false message=punto contacto alanzdo inputType=Text)
                  MoveDirectionNode (selectedDirection=ZPlus toolParams=0.1, 0.15)
                    Until DISTANCE (allowActions=false deceleration=3 distanceNodeType=STOP) Distance=0.002; motionParameters(blendRadius=0)
                  Wait Sleep waitTime=0.3
                  Set DigitalOutput pin=config_out[1]; digitalValue=1
                  Wait Sleep waitTime=0.3
                  Loop Counting (count=1) loopVariable(name=Loop_137)
                    bajar := pose_add(get_actual_tcp_pose(), bajada_broca)
                    Waypoint Waypoint (Variable): motionParameters(jointSpeed=1.047198 jointAcceleration=1.396263 cartesianSpeed=0.004 cartesianAcceleration=0.004); variable=bajar
                    subir := pose_sub(get_actual_tcp_pose(), bajada_broca)
                    MoveDirectionNode (selectedDirection=ZPlus toolParams=0.015, 0.015)
                      Until DISTANCE (allowActions=false deceleration=3 distanceNodeType=STOP) Distance=0.002; motionParameters(blendRadius=0)
                    Set DigitalOutput pin=config_out[1]; digitalValue=0
                    Waypoint Waypoint (Variable): motionParameters(jointSpeed=1.047198 jointAcceleration=1.396263 cartesianSpeed=0.015 cartesianAcceleration=0.015); variable=subir
                    bajada_broca := pose_sub(bajada_broca, bajada)
                  MoveDirectionNode (selectedDirection=ZPlus toolParams=0.03, 0.035)
                    Until DISTANCE (allowActions=false deceleration=3 distanceNodeType=STOP) Distance=0.08; motionParameters(blendRadius=0)
                  Set DigitalOutput pin=config_out[1]; digitalValue=0
                  barreno_actual := barreno_actual+1
                  SuppressedNode
                    Call Quitar_broca
                  SuppressedNode
                    Call Poner_broca
        Popup Message (haltProgram=false message=Linea17 con chica Terminada! inputType=Text)
        Folder Linea18
          Folder Marcar_puntos
            MoveL speed 100 mm/s, acceleration 500 mm/s^2 (useActiveTCP=true) feature=Base
              Waypoint Linea18_A: TCP in base x=-658.633 y=625.71 z=110.713 mm, rx=-0.2145 ry=-3.1278 rz=-0.004 rad; joints [-48.425, -62.133, 90.617, -28.11, -229.743, 0.749] deg; TCP offset x=0.411 y=-218.298 z=37.994 mm, rx=1.558 ry=-0.1255 rz=0.1212 rad
              Folder bajada_comprobacion
                MoveDirectionNode (selectedDirection=ZMinus toolParams=0.1, 0.15)
                  Until DISTANCE (allowActions=false deceleration=3 distanceNodeType=STOP) Distance=0.071; motionParameters(blendRadius=0)
                MoveDirectionNode (selectedDirection=ZMinus toolParams=0.007, 0.007)
                  Until TOOL_CONTACT_DETECTION (allowActions=false retraction=0 decelerationAcceleration=0.02 decelerationAngularAcceleration=34.906585)
                MoveDirectionNode (selectedDirection=ZPlus toolParams=0.1, 0.15)
                  Until DISTANCE (allowActions=false deceleration=3 distanceNodeType=STOP) Distance=0.08; motionParameters(blendRadius=0)
              Waypoint Linea18_AB: TCP in base x=-890.203 y=626.114 z=110.875 mm, rx=-0.2145 ry=-3.1278 rz=-0.004 rad; joints [-38.182, -44.07, 60.007, -15.504, -219.471, 0.847] deg
              SuppressedNode
                Waypoint Linea18_B: TCP in base x=-1149.588 y=625.185 z=110.393 mm, rx=1.1641 ry=-2.9058 rz=0.0105 rad; joints [-36.247, -18.765, 11.523, 7.74, -268.979, 0.895] deg; TCP offset x=0.411 y=-218.298 z=37.994 mm, rx=1.558 ry=-0.1255 rz=0.1212 rad
              Folder bajada_comprobacion
                MoveDirectionNode (selectedDirection=ZMinus toolParams=0.1, 0.15)
                  Until DISTANCE (allowActions=false deceleration=3 distanceNodeType=STOP) Distance=0.071; motionParameters(blendRadius=0)
                MoveDirectionNode (selectedDirection=ZMinus toolParams=0.007, 0.007)
                  Until TOOL_CONTACT_DETECTION (allowActions=false retraction=0 decelerationAcceleration=0.02 decelerationAngularAcceleration=34.906585)
                MoveDirectionNode (selectedDirection=ZPlus toolParams=0.1, 0.15)
                  Until DISTANCE (allowActions=false deceleration=3 distanceNodeType=STOP) Distance=0.08; motionParameters(blendRadius=0)
          Folder AB
            'desbaste_inicial'
            bajada_broca := p[0,0,-0.008,0,0,0]
            barrenos_menos1 := 9
            barreno_actual := 0
            Loop While (checkContinuously=false) expression=barreno_actual≤barrenos_menos1
              Folder Perforacion
                MoveL speed 100 mm/s, acceleration 500 mm/s^2 (useActiveTCP=true) feature=Base
                  If barreno_actual≟6
                    barreno_actual := barreno_actual+1
                  internos := interpolate_pose(Linea18_A, Linea18_AB, barreno_actual/barrenos_menos1)
                  Waypoint Waypoint (Variable): variable=internos
                  'desbaste_inicial'
                  bajada_broca := p[0,0,-0.024,0,0,0]
                  bajada := p[0,0,0.024,0,0,0]
                  MoveDirectionNode (selectedDirection=ZMinus toolParams=0.1, 0.15)
                    Until DISTANCE (allowActions=false deceleration=3 distanceNodeType=STOP) Distance=0.071; motionParameters(blendRadius=0)
                  MoveDirectionNode (selectedDirection=ZMinus toolParams=0.007, 0.007)
                    Until TOOL_CONTACT_DETECTION (allowActions=false retraction=0 decelerationAcceleration=0.02 decelerationAngularAcceleration=34.906585)
                  Popup Message (haltProgram=false message=punto contacto alanzdo inputType=Text)
                  MoveDirectionNode (selectedDirection=ZPlus toolParams=0.015, 0.015)
                    Until DISTANCE (allowActions=false deceleration=3 distanceNodeType=STOP) Distance=0.007; motionParameters(blendRadius=0)
                  Wait Sleep waitTime=0.3
                  Set DigitalOutput pin=config_out[1]; digitalValue=1
                  Wait Sleep waitTime=0.3
                  Loop Counting (count=1) loopVariable(name=Loop_139)
                    bajar := pose_add(get_actual_tcp_pose(), bajada_broca)
                    Waypoint Waypoint (Variable): motionParameters(jointSpeed=1.047198 jointAcceleration=1.396263 cartesianSpeed=0.004 cartesianAcceleration=0.004); variable=bajar
                    subir := pose_sub(get_actual_tcp_pose(), bajada_broca)
                    MoveDirectionNode (selectedDirection=ZPlus toolParams=0.015, 0.015)
                      Until DISTANCE (allowActions=false deceleration=3 distanceNodeType=STOP) Distance=0.002; motionParameters(blendRadius=0)
                    Set DigitalOutput pin=config_out[1]; digitalValue=0
                    Waypoint Waypoint (Variable): motionParameters(jointSpeed=1.047198 jointAcceleration=1.396263 cartesianSpeed=0.015 cartesianAcceleration=0.015); variable=subir
                    bajada_broca := pose_sub(bajada_broca, bajada)
                  MoveDirectionNode (selectedDirection=ZPlus toolParams=0.1, 0.15)
                    Until DISTANCE (allowActions=false deceleration=3 distanceNodeType=STOP) Distance=0.08; motionParameters(blendRadius=0)
                  Set DigitalOutput pin=config_out[1]; digitalValue=0
                  barreno_actual := barreno_actual+1
                  SuppressedNode
                    Call Quitar_broca
                  SuppressedNode
                    Call Poner_broca
        Popup Message (haltProgram=false message=Linea18 con chica Terminada! inputType=Text)
        Folder Linea18B
          Folder Marcar_puntos
            MoveL speed 100 mm/s, acceleration 500 mm/s^2 (useActiveTCP=true) feature=Base
              Waypoint Linea18_BA: TCP in base x=-915.681 y=626.148 z=110.664 mm, rx=-0.2145 ry=-3.1278 rz=-0.004 rad; joints [-37.291, -41.615, 55.578, -13.523, -218.574, 0.857] deg
              Folder bajada_comprobacion
                MoveDirectionNode (selectedDirection=ZMinus toolParams=0.1, 0.15)
                  Until DISTANCE (allowActions=false deceleration=3 distanceNodeType=STOP) Distance=0.071; motionParameters(blendRadius=0)
                MoveDirectionNode (selectedDirection=ZMinus toolParams=0.007, 0.007)
                  Until TOOL_CONTACT_DETECTION (allowActions=false retraction=0 decelerationAcceleration=0.02 decelerationAngularAcceleration=34.906585)
                MoveDirectionNode (selectedDirection=ZPlus toolParams=0.1, 0.15)
                  Until DISTANCE (allowActions=false deceleration=3 distanceNodeType=STOP) Distance=0.08; motionParameters(blendRadius=0)
              SuppressedNode
                Waypoint Linea18_AB: TCP in base x=-890.203 y=626.114 z=110.875 mm, rx=-0.2145 ry=-3.1278 rz=-0.004 rad; joints [-38.182, -44.07, 60.007, -15.504, -219.471, 0.847] deg; TCP offset x=0.411 y=-218.298 z=37.994 mm, rx=1.558 ry=-0.1255 rz=0.1212 rad
              Waypoint Linea18_B referenceName=Linea18_B: TCP in base x=-1149.588 y=625.185 z=110.393 mm, rx=1.1641 ry=-2.9058 rz=0.0105 rad; joints [-36.247, -18.765, 11.523, 7.74, -268.979, 0.895] deg; TCP offset x=0.411 y=-218.298 z=37.994 mm, rx=1.558 ry=-0.1255 rz=0.1212 rad
              Folder bajada_comprobacion
                MoveDirectionNode (selectedDirection=ZMinus toolParams=0.1, 0.15)
                  Until DISTANCE (allowActions=false deceleration=3 distanceNodeType=STOP) Distance=0.071; motionParameters(blendRadius=0)
                MoveDirectionNode (selectedDirection=ZMinus toolParams=0.007, 0.007)
                  Until TOOL_CONTACT_DETECTION (allowActions=false retraction=0 decelerationAcceleration=0.02 decelerationAngularAcceleration=34.906585)
                MoveDirectionNode (selectedDirection=ZPlus toolParams=0.1, 0.15)
                  Until DISTANCE (allowActions=false deceleration=3 distanceNodeType=STOP) Distance=0.08; motionParameters(blendRadius=0)
          Folder AB
            'desbaste_inicial'
            bajada_broca := p[0,0,-0.008,0,0,0]
            barrenos_menos1 := 9
            barreno_actual := 0
            Loop While (checkContinuously=false) expression=barreno_actual≤barrenos_menos1
              Folder Perforacion
                MoveL speed 100 mm/s, acceleration 500 mm/s^2 (useActiveTCP=true) feature=Base
                  If barreno_actual≟3
                    barreno_actual := barreno_actual+1
                  internos := interpolate_pose(Linea18_BA, Linea18_B, barreno_actual/barrenos_menos1)
                  Waypoint Waypoint (Variable): variable=internos
                  'desbaste_inicial'
                  bajada_broca := p[0,0,-0.024,0,0,0]
                  bajada := p[0,0,0.024,0,0,0]
                  MoveDirectionNode (selectedDirection=ZMinus toolParams=0.1, 0.15)
                    Until DISTANCE (allowActions=false deceleration=3 distanceNodeType=STOP) Distance=0.071; motionParameters(blendRadius=0)
                  MoveDirectionNode (selectedDirection=ZMinus toolParams=0.007, 0.007)
                    Until TOOL_CONTACT_DETECTION (allowActions=false retraction=0 decelerationAcceleration=0.02 decelerationAngularAcceleration=34.906585)
                  Popup Message (haltProgram=false message=punto contacto alanzdo inputType=Text)
                  MoveDirectionNode (selectedDirection=ZPlus toolParams=0.015, 0.015)
                    Until DISTANCE (allowActions=false deceleration=3 distanceNodeType=STOP) Distance=0.007; motionParameters(blendRadius=0)
                  Wait Sleep waitTime=0.3
                  Set DigitalOutput pin=config_out[1]; digitalValue=1
                  Wait Sleep waitTime=0.3
                  Loop Counting (count=1) loopVariable(name=Loop_28)
                    bajar := pose_add(get_actual_tcp_pose(), bajada_broca)
                    Waypoint Waypoint (Variable): motionParameters(jointSpeed=1.047198 jointAcceleration=1.396263 cartesianSpeed=0.004 cartesianAcceleration=0.004); variable=bajar
                    subir := pose_sub(get_actual_tcp_pose(), bajada_broca)
                    MoveDirectionNode (selectedDirection=ZPlus toolParams=0.015, 0.015)
                      Until DISTANCE (allowActions=false deceleration=3 distanceNodeType=STOP) Distance=0.002; motionParameters(blendRadius=0)
                    Set DigitalOutput pin=config_out[1]; digitalValue=0
                    Waypoint Waypoint (Variable): motionParameters(jointSpeed=1.047198 jointAcceleration=1.396263 cartesianSpeed=0.015 cartesianAcceleration=0.015); variable=subir
                    bajada_broca := pose_sub(bajada_broca, bajada)
                  MoveDirectionNode (selectedDirection=ZPlus toolParams=0.1, 0.15)
                    Until DISTANCE (allowActions=false deceleration=3 distanceNodeType=STOP) Distance=0.08; motionParameters(blendRadius=0)
                  Set DigitalOutput pin=config_out[1]; digitalValue=0
                  barreno_actual := barreno_actual+1
                  SuppressedNode
                    Call Quitar_broca
                  SuppressedNode
                    Call Poner_broca
        Popup Message (haltProgram=false message=Linea18B con chica Terminada! inputType=Text)
      cambiar_broca := True
      Call Quitar_broca
      Call Poner_broca
      SuppressedNode
        Folder Broca_2
          Folder Linea7
            Folder Marcar_puntos
              MoveL speed 100 mm/s, acceleration 500 mm/s^2 (useActiveTCP=true) feature=Base
                Waypoint Home2: TCP in base x=-476.229 y=0 z=568.737 mm, rx=2.0263 ry=-2.3929 rz=-0.0208 rad; joints [-32.551, -116.469, 98.413, 17.843, -302.102, -0.163] deg; TCP offset x=0.411 y=-218.298 z=37.994 mm, rx=1.558 ry=-0.1255 rz=0.1212 rad
                Waypoint Linea7_A: TCP in base x=-749.561 y=-351.839 z=110.843 mm, rx=3.1084 ry=-0.3759 rz=-0.0174 rad; joints [1.917, -65.95, 96.598, -30.808, -353.455, -0.309] deg
                Folder bajada_comprobacion
                  MoveDirectionNode (selectedDirection=ZMinus toolParams=0.1, 0.15)
                    Until DISTANCE (allowActions=false deceleration=3 distanceNodeType=STOP) Distance=0.071; motionParameters(blendRadius=0)
                  MoveDirectionNode (selectedDirection=ZMinus toolParams=0.007, 0.007)
                    Until TOOL_CONTACT_DETECTION (allowActions=false retraction=0 decelerationAcceleration=0.007 decelerationAngularAcceleration=34.906585)
                  MoveDirectionNode (selectedDirection=ZPlus toolParams=0.1, 0.15)
                    Until DISTANCE (allowActions=false deceleration=3 distanceNodeType=STOP) Distance=0.08; motionParameters(blendRadius=0)
                Waypoint Linea7_B: TCP in base x=-795.37 y=-351.638 z=110.748 mm, rx=3.1084 ry=-0.3758 rz=-0.0174 rad; joints [1.792, -62.243, 90.906, -28.822, -353.578, -0.309] deg
                Folder bajada_comprobacion
                  MoveDirectionNode (selectedDirection=ZMinus toolParams=0.1, 0.15)
                    Until DISTANCE (allowActions=false deceleration=3 distanceNodeType=STOP) Distance=0.071; motionParameters(blendRadius=0)
                  MoveDirectionNode (selectedDirection=ZMinus toolParams=0.007, 0.007)
                    Until TOOL_CONTACT_DETECTION (allowActions=false retraction=0 decelerationAcceleration=0.007 decelerationAngularAcceleration=34.906585)
                  MoveDirectionNode (selectedDirection=ZPlus toolParams=0.1, 0.15)
                    Until DISTANCE (allowActions=false deceleration=3 distanceNodeType=STOP) Distance=0.08; motionParameters(blendRadius=0)
            Folder AB
              'desbaste_inicial'
              bajada_broca := p[0,0,-0.008,0,0,0]
              barrenos_menos1 := 2
              barreno_actual := 0
              Loop While (checkContinuously=false) expression=barreno_actual≤barrenos_menos1
                Folder Perforacion
                  MoveL speed 100 mm/s, acceleration 500 mm/s^2 (useActiveTCP=true) feature=Base
                    internos := interpolate_pose(Linea7_A, Linea7_B, barreno_actual/barrenos_menos1)
                    Waypoint Waypoint (Variable): variable=internos
                    'desbaste_inicial'
                    bajada_broca := p[0,0,-0.024,0,0,0]
                    bajada := p[0,0,0.024,0,0,0]
                    MoveDirectionNode (selectedDirection=ZMinus toolParams=0.1, 0.15)
                      Until DISTANCE (allowActions=false deceleration=3 distanceNodeType=STOP) Distance=0.071; motionParameters(blendRadius=0)
                    MoveDirectionNode (selectedDirection=ZMinus toolParams=0.01, 0.01)
                      Until TOOL_CONTACT_DETECTION (allowActions=false retraction=0 decelerationAcceleration=0.01 decelerationAngularAcceleration=34.906585)
                    Popup Message (haltProgram=false message=punto contacto alanzdo inputType=Text)
                    MoveDirectionNode (selectedDirection=ZPlus toolParams=0.003, 0.005)
                      Until DISTANCE (allowActions=false deceleration=3 distanceNodeType=STOP) Distance=0.002; motionParameters(blendRadius=0)
                    Wait Sleep waitTime=0.3
                    Set DigitalOutput pin=config_out[1]; digitalValue=1
                    Wait Sleep waitTime=0.3
                    Loop Counting (count=1) loopVariable(name=Loop_47)
                      bajar := pose_add(get_actual_tcp_pose(), bajada_broca)
                      Waypoint Waypoint (Variable): motionParameters(jointSpeed=1.047198 jointAcceleration=1.396263 cartesianSpeed=0.001 cartesianAcceleration=0.005); variable=bajar
                      subir := pose_sub(get_actual_tcp_pose(), bajada_broca)
                      Waypoint Waypoint (Variable): motionParameters(jointSpeed=1.047198 jointAcceleration=1.396263 cartesianSpeed=0.005 cartesianAcceleration=0.01); variable=subir
                      bajada_broca := pose_sub(bajada_broca, bajada)
                    MoveDirectionNode (selectedDirection=ZPlus toolParams=0.1, 0.15)
                      Until DISTANCE (allowActions=false deceleration=3 distanceNodeType=STOP) Distance=0.08; motionParameters(blendRadius=0)
                    Set DigitalOutput pin=config_out[1]; digitalValue=0
                    barreno_actual := barreno_actual+1
                    Call Quitar_broca
                    Call Poner_broca
          Popup Message (haltProgram=false message=Linea7 con chica Terminada! inputType=Text)
          Folder Linea8
            Folder Marcar_puntos
              MoveL speed 100 mm/s, acceleration 500 mm/s^2 (useActiveTCP=true) feature=Base
                Waypoint Linea8_A: TCP in base x=-897.665 y=-351.421 z=110.406 mm, rx=3.1084 ry=-0.3758 rz=-0.0174 rad; joints [1.574, -53.621, 76.868, -23.4, -353.783, -0.317] deg; TCP offset x=0.411 y=-218.298 z=37.994 mm, rx=1.558 ry=-0.1255 rz=0.1212 rad
                Folder bajada_comprobacion
                  MoveDirectionNode (selectedDirection=ZMinus toolParams=0.1, 0.15)
                    Until DISTANCE (allowActions=false deceleration=3 distanceNodeType=STOP) Distance=0.071; motionParameters(blendRadius=0)
                  MoveDirectionNode (selectedDirection=ZMinus toolParams=0.007, 0.007)
                    Until TOOL_CONTACT_DETECTION (allowActions=false retraction=0 decelerationAcceleration=0.007 decelerationAngularAcceleration=34.906585)
                  MoveDirectionNode (selectedDirection=ZPlus toolParams=0.1, 0.15)
                    Until DISTANCE (allowActions=false deceleration=3 distanceNodeType=STOP) Distance=0.08; motionParameters(blendRadius=0)
                Waypoint Linea8_B: TCP in base x=-1021.743 y=-350.913 z=110.77 mm, rx=3.1084 ry=-0.3758 rz=-0.0173 rad; joints [1.351, -41.656, 55.75, -14.225, -353.984, -0.335] deg; TCP offset x=0.411 y=-218.298 z=37.994 mm, rx=1.558 ry=-0.1255 rz=0.1212 rad
                Folder bajada_comprobacion
                  MoveDirectionNode (selectedDirection=ZMinus toolParams=0.1, 0.15)
                    Until DISTANCE (allowActions=false deceleration=3 distanceNodeType=STOP) Distance=0.071; motionParameters(blendRadius=0)
                  MoveDirectionNode (selectedDirection=ZMinus toolParams=0.007, 0.007)
                    Until TOOL_CONTACT_DETECTION (allowActions=false retraction=0 decelerationAcceleration=0.007 decelerationAngularAcceleration=34.906585)
                  MoveDirectionNode (selectedDirection=ZPlus toolParams=0.1, 0.15)
                    Until DISTANCE (allowActions=false deceleration=3 distanceNodeType=STOP) Distance=0.08; motionParameters(blendRadius=0)
            Folder AB
              'desbaste_inicial'
              bajada_broca := p[0,0,-0.008,0,0,0]
              barrenos_menos1 := 5
              barreno_actual := 0
              Loop While (checkContinuously=false) expression=barreno_actual≤barrenos_menos1
                Folder Perforacion
                  MoveL speed 100 mm/s, acceleration 500 mm/s^2 (useActiveTCP=true) feature=Base
                    internos := interpolate_pose(Linea8_A, Linea8_B, barreno_actual/barrenos_menos1)
                    Waypoint Waypoint (Variable): variable=internos
                    'desbaste_inicial'
                    bajada_broca := p[0,0,-0.024,0,0,0]
                    bajada := p[0,0,0.0024,0,0,0]
                    MoveDirectionNode (selectedDirection=ZMinus toolParams=0.1, 0.15)
                      Until DISTANCE (allowActions=false deceleration=3 distanceNodeType=STOP) Distance=0.071; motionParameters(blendRadius=0)
                    MoveDirectionNode (selectedDirection=ZMinus toolParams=0.01, 0.01)
                      Until TOOL_CONTACT_DETECTION (allowActions=false retraction=0 decelerationAcceleration=0.01 decelerationAngularAcceleration=34.906585)
                    Popup Message (haltProgram=false message=punto contacto alanzdo inputType=Text)
                    MoveDirectionNode (selectedDirection=ZPlus toolParams=0.003, 0.005)
                      Until DISTANCE (allowActions=false deceleration=3 distanceNodeType=STOP) Distance=0.002; motionParameters(blendRadius=0)
                    Wait Sleep waitTime=0.3
                    Set DigitalOutput pin=config_out[1]; digitalValue=1
                    Wait Sleep waitTime=0.3
                    Loop Counting (count=1) loopVariable(name=Loop_53)
                      bajar := pose_add(get_actual_tcp_pose(), bajada_broca)
                      Waypoint Waypoint (Variable): motionParameters(jointSpeed=1.047198 jointAcceleration=1.396263 cartesianSpeed=0.001 cartesianAcceleration=0.005); variable=bajar
                      subir := pose_sub(get_actual_tcp_pose(), bajada_broca)
                      Waypoint Waypoint (Variable): motionParameters(jointSpeed=1.047198 jointAcceleration=1.396263 cartesianSpeed=0.005 cartesianAcceleration=0.01); variable=subir
                      bajada_broca := pose_sub(bajada_broca, bajada)
                    MoveDirectionNode (selectedDirection=ZPlus toolParams=0.1, 0.15)
                      Until DISTANCE (allowActions=false deceleration=3 distanceNodeType=STOP) Distance=0.08; motionParameters(blendRadius=0)
                    Set DigitalOutput pin=config_out[1]; digitalValue=0
                    barreno_actual := barreno_actual+1
                    Call Quitar_broca
                    Call Poner_broca
          Popup Message (haltProgram=false message=Linea8 con chica Terminada! inputType=Text)
          Folder Linea9
            Folder Marcar_puntos
              MoveL speed 100 mm/s, acceleration 500 mm/s^2 (useActiveTCP=true) feature=Base
                Waypoint Linea9_A: TCP in base x=-1101.64 y=-350.63 z=110.828 mm, rx=3.1084 ry=-0.3759 rz=-0.0174 rad; joints [1.234, -31.471, 36.669, -5.317, -354.073, -0.351] deg; TCP offset x=0.411 y=-218.298 z=37.994 mm, rx=1.558 ry=-0.1255 rz=0.1212 rad
                Folder bajada_comprobacion
                  MoveDirectionNode (selectedDirection=ZMinus toolParams=0.1, 0.15)
                    Until DISTANCE (allowActions=false deceleration=3 distanceNodeType=STOP) Distance=0.071; motionParameters(blendRadius=0)
                  MoveDirectionNode (selectedDirection=ZMinus toolParams=0.007, 0.007)
                    Until TOOL_CONTACT_DETECTION (allowActions=false retraction=0 decelerationAcceleration=0.007 decelerationAngularAcceleration=34.906585)
                  MoveDirectionNode (selectedDirection=ZPlus toolParams=0.1, 0.15)
                    Until DISTANCE (allowActions=false deceleration=3 distanceNodeType=STOP) Distance=0.08; motionParameters(blendRadius=0)
                Waypoint Linea9_B: TCP in base x=-1151.202 y=-350.816 z=110.405 mm, rx=3.1084 ry=-0.3759 rz=-0.0174 rad; joints [1.184, -21.077, 16.327, 4.623, -354.093, -0.341] deg
                Folder bajada_comprobacion
                  MoveDirectionNode (selectedDirection=ZMinus toolParams=0.1, 0.15)
                    Until DISTANCE (allowActions=false deceleration=3 distanceNodeType=STOP) Distance=0.071; motionParameters(blendRadius=0)
                  MoveDirectionNode (selectedDirection=ZMinus toolParams=0.007, 0.007)
                    Until TOOL_CONTACT_DETECTION (allowActions=false retraction=0 decelerationAcceleration=0.007 decelerationAngularAcceleration=34.906585)
                  MoveDirectionNode (selectedDirection=ZPlus toolParams=0.1, 0.15)
                    Until DISTANCE (allowActions=false deceleration=3 distanceNodeType=STOP) Distance=0.08; motionParameters(blendRadius=0)
            Folder AB
              'desbaste_inicial'
              bajada_broca := p[0,0,-0.008,0,0,0]
              barrenos_menos1 := 2
              barreno_actual := 0
              Loop While (checkContinuously=false) expression=barreno_actual≤barrenos_menos1
                Folder Perforacion
                  MoveL speed 100 mm/s, acceleration 500 mm/s^2 (useActiveTCP=true) feature=Base
                    internos := interpolate_pose(Linea9_A, Linea9_B, barreno_actual/barrenos_menos1)
                    Waypoint Waypoint (Variable): variable=internos
                    'desbaste_inicial'
                    bajada_broca := p[0,0,-0.024,0,0,0]
                    bajada := p[0,0,0.024,0,0,0]
                    MoveDirectionNode (selectedDirection=ZMinus toolParams=0.1, 0.15)
                      Until DISTANCE (allowActions=false deceleration=3 distanceNodeType=STOP) Distance=0.071; motionParameters(blendRadius=0)
                    MoveDirectionNode (selectedDirection=ZMinus toolParams=0.01, 0.01)
                      Until TOOL_CONTACT_DETECTION (allowActions=false retraction=0 decelerationAcceleration=0.01 decelerationAngularAcceleration=34.906585)
                    Popup Message (haltProgram=false message=punto contacto alanzdo inputType=Text)
                    MoveDirectionNode (selectedDirection=ZPlus toolParams=0.003, 0.005)
                      Until DISTANCE (allowActions=false deceleration=3 distanceNodeType=STOP) Distance=0.002; motionParameters(blendRadius=0)
                    Wait Sleep waitTime=0.3
                    Set DigitalOutput pin=config_out[1]; digitalValue=1
                    Wait Sleep waitTime=0.3
                    Loop Counting (count=1) loopVariable=Loop_56
                      bajar := pose_add(get_actual_tcp_pose(), bajada_broca)
                      Waypoint Waypoint (Variable): motionParameters(jointSpeed=1.047198 jointAcceleration=1.396263 cartesianSpeed=0.001 cartesianAcceleration=0.005); variable=bajar
                      subir := pose_sub(get_actual_tcp_pose(), bajada_broca)
                      Waypoint Waypoint (Variable): motionParameters(jointSpeed=1.047198 jointAcceleration=1.396263 cartesianSpeed=0.005 cartesianAcceleration=0.01); variable=subir
                      bajada_broca := pose_sub(bajada_broca, bajada)
                    MoveDirectionNode (selectedDirection=ZPlus toolParams=0.1, 0.15)
                      Until DISTANCE (allowActions=false deceleration=3 distanceNodeType=STOP) Distance=0.08; motionParameters(blendRadius=0)
                    Set DigitalOutput pin=config_out[1]; digitalValue=0
                    barreno_actual := barreno_actual+1
                    Call Quitar_broca
                    Call Poner_broca
          Popup Message (haltProgram=false message=Linea9 con chica Terminada! inputType=Text)
          Folder Linea10
            Folder Marcar_puntos
              MoveL speed 100 mm/s, acceleration 500 mm/s^2 (useActiveTCP=true) feature=Base
                Waypoint Home2: TCP in base x=-476.229 y=0 z=568.737 mm, rx=2.0263 ry=-2.3929 rz=-0.0208 rad; joints [-32.551, -116.469, 98.413, 17.843, -302.102, -0.163] deg; TCP offset x=0.411 y=-218.298 z=37.994 mm, rx=1.558 ry=-0.1255 rz=0.1212 rad
                Waypoint Linea10_A: TCP in base x=-633.044 y=-316.972 z=110.617 mm, rx=3.1084 ry=-0.3759 rz=-0.0173 rad; joints [-0.95, -76.145, 111.037, -35.154, -356.326, -0.202] deg; TCP offset x=0.411 y=-218.298 z=37.994 mm, rx=1.558 ry=-0.1255 rz=0.1212 rad
                Folder bajada_comprobacion
                  MoveDirectionNode (selectedDirection=ZMinus toolParams=0.1, 0.15)
                    Until DISTANCE (allowActions=false deceleration=3 distanceNodeType=STOP) Distance=0.071; motionParameters(blendRadius=0)
                  MoveDirectionNode (selectedDirection=ZMinus toolParams=0.007, 0.007)
                    Until TOOL_CONTACT_DETECTION (allowActions=false retraction=0 decelerationAcceleration=0.007 decelerationAngularAcceleration=34.906585)
                  MoveDirectionNode (selectedDirection=ZPlus toolParams=0.1, 0.15)
                    Until DISTANCE (allowActions=false deceleration=3 distanceNodeType=STOP) Distance=0.08; motionParameters(blendRadius=0)
                Waypoint Linea10_B: TCP in base x=-636.724 y=-267.195 z=110.576 mm, rx=2.0205 ry=-2.3939 rz=-0.0206 rad; joints [10.728, -83.916, 120.692, -37.175, -258.773, -0.177] deg
                Folder bajada_comprobacion
                  MoveDirectionNode (selectedDirection=ZMinus toolParams=0.1, 0.15)
                    Until DISTANCE (allowActions=false deceleration=3 distanceNodeType=STOP) Distance=0.071; motionParameters(blendRadius=0)
                  MoveDirectionNode (selectedDirection=ZMinus toolParams=0.007, 0.007)
                    Until TOOL_CONTACT_DETECTION (allowActions=false retraction=0 decelerationAcceleration=0.007 decelerationAngularAcceleration=34.906585)
                  MoveDirectionNode (selectedDirection=ZPlus toolParams=0.1, 0.15)
                    Until DISTANCE (allowActions=false deceleration=3 distanceNodeType=STOP) Distance=0.08; motionParameters(blendRadius=0)
            Folder AB
              'desbaste_inicial'
              bajada_broca := p[0,0,-0.008,0,0,0]
              barrenos_menos1 := 2
              barreno_actual := 0
              Loop While (checkContinuously=false) expression=barreno_actual≤barrenos_menos1
                Folder Perforacion
                  MoveL speed 100 mm/s, acceleration 500 mm/s^2 (useActiveTCP=true) feature=Base
                    internos := interpolate_pose(Linea10_A, Linea10_B, barreno_actual/barrenos_menos1)
                    Waypoint Waypoint (Variable): variable=internos
                    'desbaste_inicial'
                    bajada_broca := p[0,0,-0.024,0,0,0]
                    bajada := p[0,0,0.024,0,0,0]
                    MoveDirectionNode (selectedDirection=ZMinus toolParams=0.1, 0.15)
                      Until DISTANCE (allowActions=false deceleration=3 distanceNodeType=STOP) Distance=0.071; motionParameters(blendRadius=0)
                    MoveDirectionNode (selectedDirection=ZMinus toolParams=0.001, 0.001)
                      Until TOOL_CONTACT_DETECTION (allowActions=false retraction=0 decelerationAcceleration=0.001 decelerationAngularAcceleration=34.906585)
                    Popup Message (haltProgram=false message=punto contacto alanzdo inputType=Text)
                    MoveDirectionNode (selectedDirection=ZPlus toolParams=0.003, 0.005)
                      Until DISTANCE (allowActions=false deceleration=3 distanceNodeType=STOP) Distance=0.002; motionParameters(blendRadius=0)
                    Wait Sleep waitTime=0.3
                    Set DigitalOutput pin=config_out[1]; digitalValue=1
                    Wait Sleep waitTime=0.3
                    Loop Counting (count=1) loopVariable(name=Loop_58)
                      bajar := pose_add(get_actual_tcp_pose(), bajada_broca)
                      Waypoint Waypoint (Variable): motionParameters(jointSpeed=1.047198 jointAcceleration=1.396263 cartesianSpeed=0.001 cartesianAcceleration=0.005); variable=bajar
                      subir := pose_sub(get_actual_tcp_pose(), bajada_broca)
                      Waypoint Waypoint (Variable): motionParameters(jointSpeed=1.047198 jointAcceleration=1.396263 cartesianSpeed=0.005 cartesianAcceleration=0.01); variable=subir
                      bajada_broca := pose_sub(bajada_broca, bajada)
                    MoveDirectionNode (selectedDirection=ZPlus toolParams=0.1, 0.15)
                      Until DISTANCE (allowActions=false deceleration=3 distanceNodeType=STOP) Distance=0.08; motionParameters(blendRadius=0)
                    Set DigitalOutput pin=config_out[1]; digitalValue=0
                    barreno_actual := barreno_actual+1
                    Call Quitar_broca
                    Call Poner_broca
          Popup Message (haltProgram=false message=Linea10 con chica Terminada! inputType=Text)
          Folder Linea11
            Folder Marcar_puntos
              MoveL speed 100 mm/s, acceleration 500 mm/s^2 (useActiveTCP=true) feature=Base
                Waypoint Linea11_A: TCP in base x=-636.133 y=-137.915 z=110.44 mm, rx=2.0204 ry=-2.394 rz=-0.0205 rad; joints [-4.201, -88.707, 125.915, -37.584, -273.698, -0.078] deg
                Folder bajada_comprobacion
                  MoveDirectionNode (selectedDirection=ZMinus toolParams=0.1, 0.15)
                    Until DISTANCE (allowActions=false deceleration=3 distanceNodeType=STOP) Distance=0.071; motionParameters(blendRadius=0)
                  MoveDirectionNode (selectedDirection=ZMinus toolParams=0.007, 0.007)
                    Until TOOL_CONTACT_DETECTION (allowActions=false retraction=0 decelerationAcceleration=0.007 decelerationAngularAcceleration=34.906585)
                  MoveDirectionNode (selectedDirection=ZPlus toolParams=0.1, 0.15)
                    Until DISTANCE (allowActions=false deceleration=3 distanceNodeType=STOP) Distance=0.08; motionParameters(blendRadius=0)
                Waypoint Linea11_B: TCP in base x=-635.407 y=-82.609 z=110.403 mm, rx=2.0204 ry=-2.3939 rz=-0.0206 rad; joints [-11.006, -90.015, 127.249, -37.609, -280.504, -0.032] deg
                Folder bajada_comprobacion
                  MoveDirectionNode (selectedDirection=ZMinus toolParams=0.1, 0.15)
                    Until DISTANCE (allowActions=false deceleration=3 distanceNodeType=STOP) Distance=0.071; motionParameters(blendRadius=0)
                  MoveDirectionNode (selectedDirection=ZMinus toolParams=0.007, 0.007)
                    Until TOOL_CONTACT_DETECTION (allowActions=false retraction=0 decelerationAcceleration=0.007 decelerationAngularAcceleration=34.906585)
                  MoveDirectionNode (selectedDirection=ZPlus toolParams=0.1, 0.15)
                    Until DISTANCE (allowActions=false deceleration=3 distanceNodeType=STOP) Distance=0.08; motionParameters(blendRadius=0)
            Folder AB
              'desbaste_inicial'
              bajada_broca := p[0,0,-0.008,0,0,0]
              barrenos_menos1 := 2
              barreno_actual := 0
              Loop While (checkContinuously=false) expression=barreno_actual≤barrenos_menos1
                Folder Perforacion
                  MoveL speed 100 mm/s, acceleration 500 mm/s^2 (useActiveTCP=true) feature=Base
                    SuppressedNode
                      If barreno_actual≟5
                        barreno_actual := barreno_actual+1
                    internos := interpolate_pose(Linea11_A, Linea11_B, barreno_actual/barrenos_menos1)
                    Waypoint Waypoint (Variable): variable=internos
                    'desbaste_inicial'
                    bajada_broca := p[0,0,-0.024,0,0,0]
                    bajada := p[0,0,0.024,0,0,0]
                    MoveDirectionNode (selectedDirection=ZMinus toolParams=0.1, 0.15)
                      Until DISTANCE (allowActions=false deceleration=3 distanceNodeType=STOP) Distance=0.071; motionParameters(blendRadius=0)
                    MoveDirectionNode (selectedDirection=ZMinus toolParams=0.001, 0.001)
                      Until TOOL_CONTACT_DETECTION (allowActions=false retraction=0 decelerationAcceleration=0.001 decelerationAngularAcceleration=34.906585)
                    Popup Message (haltProgram=false message=punto contacto alanzdo inputType=Text)
                    MoveDirectionNode (selectedDirection=ZPlus toolParams=0.003, 0.005)
                      Until DISTANCE (allowActions=false deceleration=3 distanceNodeType=STOP) Distance=0.002; motionParameters(blendRadius=0)
                    Wait Sleep waitTime=0.3
                    Set DigitalOutput pin=config_out[1]; digitalValue=1
                    Wait Sleep waitTime=0.3
                    Loop Counting (count=1) loopVariable=Loop_74
                      bajar := pose_add(get_actual_tcp_pose(), bajada_broca)
                      Waypoint Waypoint (Variable): motionParameters(jointSpeed=1.047198 jointAcceleration=1.396263 cartesianSpeed=0.001 cartesianAcceleration=0.005); variable=bajar
                      subir := pose_sub(get_actual_tcp_pose(), bajada_broca)
                      Waypoint Waypoint (Variable): motionParameters(jointSpeed=1.047198 jointAcceleration=1.396263 cartesianSpeed=0.005 cartesianAcceleration=0.01); variable=subir
                      bajada_broca := pose_sub(bajada_broca, bajada)
                    MoveDirectionNode (selectedDirection=ZPlus toolParams=0.1, 0.15)
                      Until DISTANCE (allowActions=false deceleration=3 distanceNodeType=STOP) Distance=0.08; motionParameters(blendRadius=0)
                    Set DigitalOutput pin=config_out[1]; digitalValue=0
                    barreno_actual := barreno_actual+1
                    Call Quitar_broca
                    Call Poner_broca
          Popup Message (haltProgram=false message=Linea11 con chica Terminada! inputType=Text)
          Folder Linea12
            Folder Marcar_puntos
              MoveL speed 100 mm/s, acceleration 500 mm/s^2 (useActiveTCP=true) feature=Base
                Waypoint Linea12_A: TCP in base x=-635.979 y=-59.028 z=110.553 mm, rx=2.0204 ry=-2.3939 rz=-0.0205 rad; joints [-13.896, -90.321, 127.534, -37.586, -283.394, -0.016] deg
                Folder bajada_comprobacion
                  MoveDirectionNode (selectedDirection=ZMinus toolParams=0.1, 0.15)
                    Until DISTANCE (allowActions=false deceleration=3 distanceNodeType=STOP) Distance=0.071; motionParameters(blendRadius=0)
                  MoveDirectionNode (selectedDirection=ZMinus toolParams=0.007, 0.007)
                    Until TOOL_CONTACT_DETECTION (allowActions=false retraction=0 decelerationAcceleration=0.007 decelerationAngularAcceleration=34.906585)
                  MoveDirectionNode (selectedDirection=ZPlus toolParams=0.1, 0.15)
                    Until DISTANCE (allowActions=false deceleration=3 distanceNodeType=STOP) Distance=0.08; motionParameters(blendRadius=0)
                Waypoint Linea12_B: TCP in base x=-634.713 y=114.271 z=110.459 mm, rx=2.0204 ry=-2.3939 rz=-0.0206 rad; joints [-33.928, -89.524, 126.748, -37.639, -303.428, 0.135] deg
                Folder bajada_comprobacion
                  MoveDirectionNode (selectedDirection=ZMinus toolParams=0.1, 0.15)
                    Until DISTANCE (allowActions=false deceleration=3 distanceNodeType=STOP) Distance=0.071; motionParameters(blendRadius=0)
                  MoveDirectionNode (selectedDirection=ZMinus toolParams=0.007, 0.007)
                    Until TOOL_CONTACT_DETECTION (allowActions=false retraction=0 decelerationAcceleration=0.007 decelerationAngularAcceleration=34.906585)
                  MoveDirectionNode (selectedDirection=ZPlus toolParams=0.1, 0.15)
                    Until DISTANCE (allowActions=false deceleration=3 distanceNodeType=STOP) Distance=0.08; motionParameters(blendRadius=0)
            Folder AB
              'desbaste_inicial'
              bajada_broca := p[0,0,-0.008,0,0,0]
              barrenos_menos1 := 7
              barreno_actual := 0
              Loop While (checkContinuously=false) expression=barreno_actual≤barrenos_menos1
                Folder Perforacion
                  MoveL speed 100 mm/s, acceleration 500 mm/s^2 (useActiveTCP=true) feature=Base
                    If barreno_actual≟2
                      barreno_actual := barreno_actual+1
                    internos := interpolate_pose(Linea12_A, Linea12_B, barreno_actual/barrenos_menos1)
